# B&R Automation Studio project A2019059_Linka_Power_CP
Automation Studio 4.10.3.60 SP; technology packages: mapp 5.15.0, mappCockpit 5.15.0, mappMotion 5.15.1, mappView 5.15.1

## Configuration Config1

CPU 5PC900.TS17-00, AutomationRuntime B4.91, Build 6.3.0, Safety 1.10, Vc 

### Task classes (Cpu.sw)
```
Cyclic#1 (cycle 4000 us, tolerance 0 us):
  RiadenieSe <- RiadenieServ.RiadenieServ.prg
  P1_Skrutk1 <- Program.Pracovisko_1.P1_SkrutkovaciSet_M5.prg
  P1_Skrutk2 <- Program.Pracovisko_1.P1_SkrutkovaciSet_M4.prg
  P1_Skrutko <- Program.Pracovisko_1.P1_SkrutkovaciSet_K30.prg
  P2_Skrutko <- Program.Pracovisko_2.P2_SkrutkovaciSet_MaticaM4.prg
  P2_Skrutk2 <- Program.Pracovisko_2.P2_SkrutkovaciSet_M5.prg
  P2_Skrutk3 <- Program.Pracovisko_2.P2_SkrutkovaciSet_M6.prg
  P2_Skrutk1 <- Program.Pracovisko_2.P2_SkrutkovaciSet_M4.prg
  P3_Skrutk1 <- Program.Pracovisko_3.P3_SkrutkovaciSet_M5.prg
  P3_Skrutko <- Program.Pracovisko_3.P3_SkrutkovaciSet_K40.prg
  CAM_12 <- (binary)
  CAM_11 <- (binary)
  CAM_14 <- (binary)
  CAM_5 <- (binary)
  CAM_7 <- (binary)
  CAM_1 <- (binary)
  CAM_3 <- (binary)
  CAM_2 <- (binary)
  CAM_9 <- (binary)
  CAM_8 <- (binary)
  CAM_10 <- (binary)
  CAM_17 <- (binary)
  CAM_4 <- (binary)
  CAM_6 <- (binary)
  CAM_13 <- (binary)
  CAM_16 <- (binary)
  CAM_15 <- (binary)
  CAM1 <- (binary)
Cyclic#2 (cycle 8000 us, tolerance 0 us):
  TaktimePra <- MeranieTaktimePracovisk.TaktimeVytah_ST1.prg
  TaktimeSro <- MeranieTaktimePracovisk.TaktimeSrobovanie_ST2.prg
  TaktimeZak <- MeranieTaktimePracovisk.TaktimeZaklTesnenia_ST3.prg
  TaktimeMat <- MeranieTaktimePracovisk.TaktimeMaticovacka_ST4.prg
  TaktimeSr1 <- MeranieTaktimePracovisk.TaktimeSrobovanie_ST5.prg
  TaktimeZva <- MeranieTaktimePracovisk.TaktimeZvaranie_ST6.prg
  Taktime_Sr <- MeranieTaktimePracovisk.Taktime_Srobovanie_ST7.prg
  Taktime_Le <- MeranieTaktimePracovisk.Taktime_LeakageTestA_ST8A.prg
  Taktime_L1 <- MeranieTaktimePracovisk.Taktime_LeakageTestB_ST8B.prg
  Taktime_Fu <- MeranieTaktimePracovisk.Taktime_FunkcnyTestA_ST9A.prg
  Taktime_F1 <- MeranieTaktimePracovisk.Taktime_FunkcnyTestB_ST9B.prg
  Taktime_Et <- MeranieTaktimePracovisk.Taktime_Etiketovacka_ST9.prg
  Taktime_Vy <- MeranieTaktimePracovisk.Taktime_Vytah_ST10.prg
  FTP_CAM1 <- OdosielanieFotiek.FTP_CAM1.prg
  FTP_CAM2 <- OdosielanieFotiek.FTP_CAM2.prg
  FTP_CAM4 <- OdosielanieFotiek.FTP_CAM4.prg
  FTP_CAM6 <- OdosielanieFotiek.FTP_CAM6.prg
  FTP_CAM9 <- OdosielanieFotiek.FTP_CAM9.prg
  FTP_CAM10 <- OdosielanieFotiek.FTP_CAM10.prg
  FTP_CAM11 <- OdosielanieFotiek.FTP_CAM11.prg
  FTP_CAM12 <- OdosielanieFotiek.FTP_CAM12.prg
  FTP_CAM13 <- OdosielanieFotiek.FTP_CAM13.prg
  FTP_CAM15 <- OdosielanieFotiek.FTP_CAM15.prg
  FTP_CAM16 <- OdosielanieFotiek.FTP_CAM16.prg
  FTP_CAM17 <- OdosielanieFotiek.FTP_CAM17.prg
  FTP_DMP_CA <- OdosielanieFotiek.FTP_DMP_CAM1.prg
  FTP_DMP_C1 <- OdosielanieFotiek.FTP_DMP_CAM2.prg
  FTP_DMP_C2 <- OdosielanieFotiek.FTP_DMP_CAM3.prg
  FTP_DMP_C3 <- OdosielanieFotiek.FTP_DMP_CAM4.prg
  FTP_DMP_C4 <- OdosielanieFotiek.FTP_DMP_CAM5.prg
  FTP_DMP_C5 <- OdosielanieFotiek.FTP_DMP_CAM6.prg
  FTP_DMP_C6 <- OdosielanieFotiek.FTP_DMP_CAM7.prg
  FTP_DMP_C7 <- OdosielanieFotiek.FTP_DMP_CAM8.prg
  FTP_DMP_C8 <- OdosielanieFotiek.FTP_DMP_CAM9.prg
  FTP_DMP_C9 <- OdosielanieFotiek.FTP_DMP_CAM10.prg
  FTP_DMP_10 <- OdosielanieFotiek.FTP_DMP_CAM11.prg
  FTP_DMP_11 <- OdosielanieFotiek.FTP_DMP_CAM12.prg
  FTP_DMP_12 <- OdosielanieFotiek.FTP_DMP_CAM13.prg
  FTP_DMP_13 <- OdosielanieFotiek.FTP_DMP_CAM14.prg
  FTP_DMP_14 <- OdosielanieFotiek.FTP_DMP_CAM15.prg
  FTP_DMP_15 <- OdosielanieFotiek.FTP_DMP_CAM16.prg
  FTP_DMP_16 <- OdosielanieFotiek.FTP_DMP_CAM17.prg
  Users_Pane <- Uzivatelia.Users_Panel1.prg
  Users_Pan1 <- Uzivatelia.Users_Panel2.prg
  Program12 <- Uzivatelia.Users_Panel3.prg
  Users_Main <- Uzivatelia.Users_Main.prg
Cyclic#3 (cycle 48000 us, tolerance 48000 us):
  P1_Vytah_S <- TracebilitySystem.P1_Vytah_ST1.prg
  Program2 <- TracebilitySystem.P1_Srobovanie_ST2.prg
  Program3 <- TracebilitySystem.P2_ZakladacTesnenia_ST3.prg
  Program4 <- TracebilitySystem.P2_Maticovacka_ST4.prg
  Program5 <- TracebilitySystem.P2_Srobovanie_ST5.prg
  Program6 <- TracebilitySystem.P2_Zvaranie_ST6.prg
  Program7 <- TracebilitySystem.P3_Srobovanie_ST7.prg
  Program8 <- TracebilitySystem.P3_LeakageTestA_ST8A.prg
  Program9 <- TracebilitySystem.P3_LeakageTestB_ST8B.prg
  Program10 <- TracebilitySystem.P4_Etiketovacka_ST9.prg
  Program11 <- TracebilitySystem.P4_Vytah_ST10.prg
  LimitneSni <- RiadenieServ.LimitneSnimace.prg
  P4_StoperF <- Program.Pracovisko_4.P4_StoperFunkcnyTestA.prg
  P4_Stoper1 <- Program.Pracovisko_4.P4_StoperFunkcnyTestB.prg
  P3_Srobova <- Program.Pracovisko_3.P3_Srobovanie.prg
  Blikanie10 <- Blikace.Blikanie100ms.prg
Cyclic#4:
  Blikanie20 <- Blikace.Blikanie200ms.prg
  RFID_Prg <- Uzivatelia.RFID_Prg.prg
  P1_Main <- Program.Pracovisko_1.P1_Main.prg
  P1_Dopravn <- Program.Pracovisko_1.P1_Dopravniky.prg
  P1_SpodnyS <- Program.Pracovisko_1.P1_SpodnyStoper.prg
  P1_Akumula <- Program.Pracovisko_1.P1_AkumulacnyStoper.prg
  P1_Ovlada1 <- Program.Pracovisko_1.P1_OvladanieSafety.prg
  P2_Main <- Program.Pracovisko_2.P2_Main.prg
  P2_Dopravn <- Program.Pracovisko_2.P2_Dopravniky.prg
  P2_Akumula <- Program.Pracovisko_3.P3_VstupnyStoper.prg
  P2_Ovlada1 <- Program.Pracovisko_2.P2_OvladanieSafety.prg
  P3_Main <- Program.Pracovisko_3.P3_Main.prg
  P3_Dopravn <- Program.Pracovisko_3.P3_Dopravniky.prg
  P3_SpodnyS <- Program.Pracovisko_3.P3_SpodnyStoper.prg
  P3_Akumula <- Program.Pracovisko_3.P3_AkumulacnyStoper.prg
  P3_Ovlada1 <- Program.Pracovisko_3.P3_OvladanieSafety.prg
  P4_Main <- Program.Pracovisko_4.P4_Main.prg
  P4_Dopravn <- Program.Pracovisko_4.P4_Dopravniky.prg
  P4_Ovlada1 <- Program.Pracovisko_4.P4_OvladanieSafety.prg
  DatumCasPL <- DatumCasPLC.DatumCasPLC.prg
  Main <- Program.Linka.Main.prg
  OvladanieS <- Program.Linka.OvladanieSafety.prg
  UkladacieB <- UkladacieBuffery.UkladacieBuffery.prg
Cyclic#5 (cycle 248000 us, tolerance 248000 us):
  P1_Ovlada2 <- Program.Linka.OvladanieVizu.prg
  P1_Ovladan <- Program.Pracovisko_1.P1_OvladanieVizu.prg
  P2_Ovladan <- Program.Pracovisko_2.P2_OvladanieVizu.prg
  P3_Ovladan <- Program.Pracovisko_3.P34_OvladanieVizu.prg
  P1_Remanen <- RemanentnePremenne.P1_RemanentnePremenne.prg
  Remanentne <- RemanentnePremenne.P2_RemanentnePremenne.prg
  P34_Remane <- RemanentnePremenne.P34_RemanentnePremenne.prg
  Blikanie50 <- Blikace.Blikanie500ms.prg
Cyclic#6:
  Blikanie1s <- Blikace.Blikanie1s.prg
Cyclic#8 (cycle 8000 us, tolerance 8000 us):
  P1_Alarmy <- Alarmy.P1_Alarmy.prg
  P2_Alarmy <- Alarmy.P2_Alarmy.prg
  P34_Alarmy <- Alarmy.P34_Alarmy.prg
  P1_Vytah <- Program.Pracovisko_1.P1_Vytah.prg
  P1_Srobova <- Program.Pracovisko_1.P1_Srobovanie.prg
  P1_StoperS <- Program.Pracovisko_1.P1_StoperSrobovania.prg
  P1_Robot <- Program.Pracovisko_1.P1_Robot.prg
  P2_Zaklada <- Program.Pracovisko_2.P2_ZakladacTesnenia.prg
  P2_StoperZ <- Program.Pracovisko_2.P2_StoperZaklTesnenia.prg
  P2_StoperM <- Program.Pracovisko_2.P2_StoperMaticovacky.prg
  P2_Srobova <- Program.Pracovisko_2.P2_Srobovanie.prg
  P2_StoperS <- Program.Pracovisko_2.P2_StoperSrobovania.prg
  P2_Robot <- Program.Pracovisko_2.P2_Robot.prg
  P2_Zvarani <- Program.Pracovisko_2.P2_Zvaranie.prg
  P2_Cisteni <- Program.Pracovisko_2.P2_Cistenie.prg
  P2_Stoper1 <- Program.Pracovisko_2.P2_StoperZvarania.prg
  P3_StoperS <- Program.Pracovisko_3.P3_StoperSrobovania.prg
  P3_StoperL <- Program.Pracovisko_3.P3_StoperLeakageTestA.prg
  P3_Stoper1 <- Program.Pracovisko_3.P3_StoperLeakageTestB.prg
  P4_StoperE <- Program.Pracovisko_4.P4_StoperEtiketovacky.prg
  P4_Vytah <- Program.Pracovisko_4.P4_Vytah.prg
DataObjects: McAcpSys, assl1
Binaries: arsvcreg, udbdef, mvLoader, TCData, FWRules, mCoWebSc, mcacpdrv, McAcpSim, mcprofgen, TCLang, arflatprv, arcoal, ashwd, ashwac, Settings, User, sysconf, asfw, arconfig, asnxdb1, iomap, Role, Config_3, Config_1, Config, Config_2, Config_4, Config_5, Config_6, Config_7, Config_8, Config_9, Config_15, Config_14, TC, asiol4, asiol10, asiol3, asiol1, asiol2, Config_20, Config_19, Config_18, asiol5, Config_21, asiol6, asiol7, Config_23, Config_22, asiol9, asiol8, Config_10, asnxdb2, TraceConfi, Users, Config_13, Config_11, Config_12, Config_17, Config_16, asnxdb3
Libraries: CoTrace, AsZip, FileIO, runtime, AsBrStr, sys_lib, dvframe, AsUSB, standard, asstring, SC, AxisLib, MpBase, MpAlarmX, astime, MpRecipe, AsSafety, DataObj, AsXml, MpServer, AsBrWStr, AsIODiag, AsHttp, AsMem, AsMath, AsTCP, AsIecCon, IecCheck, MpAxis, McAxis, McBase, McAcpAx, McStpAx, McAcpPar, AtlasCopco, SKTcp, RFID, asio, asioacc, powerlnk, aruser, arssl, asepl, aseth, ashw, arcert
```

### Hardware
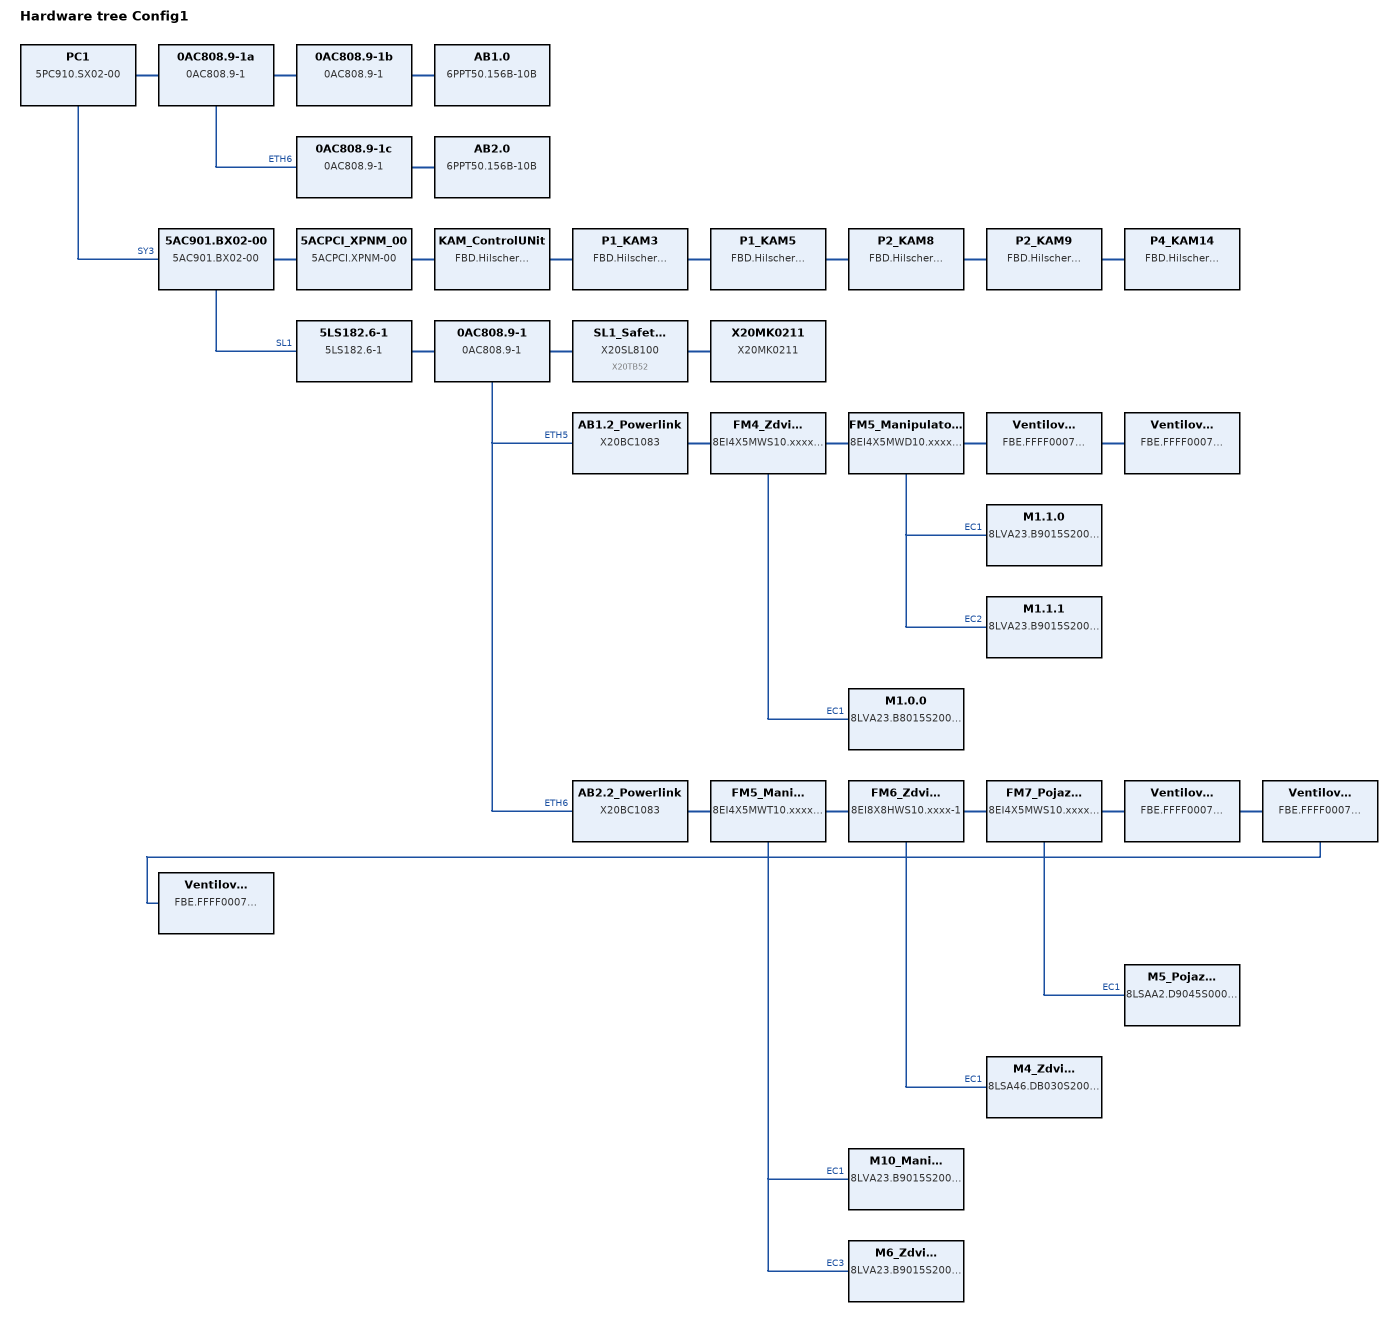
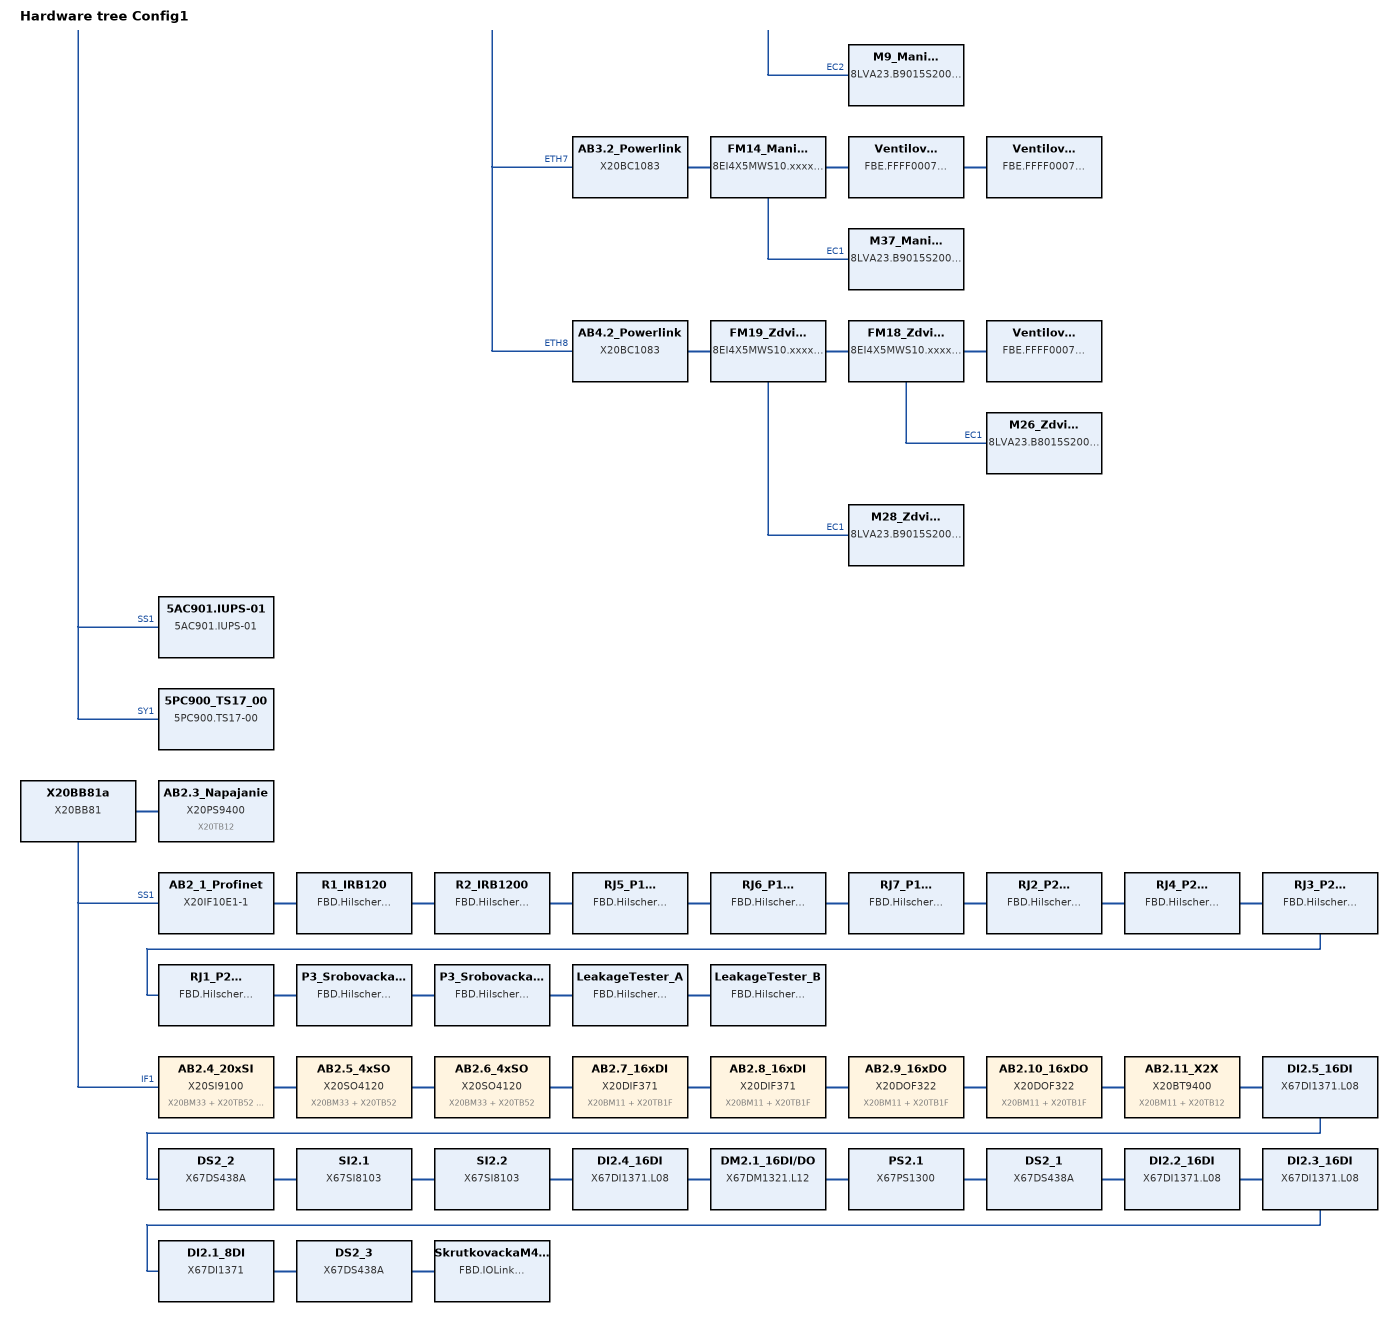
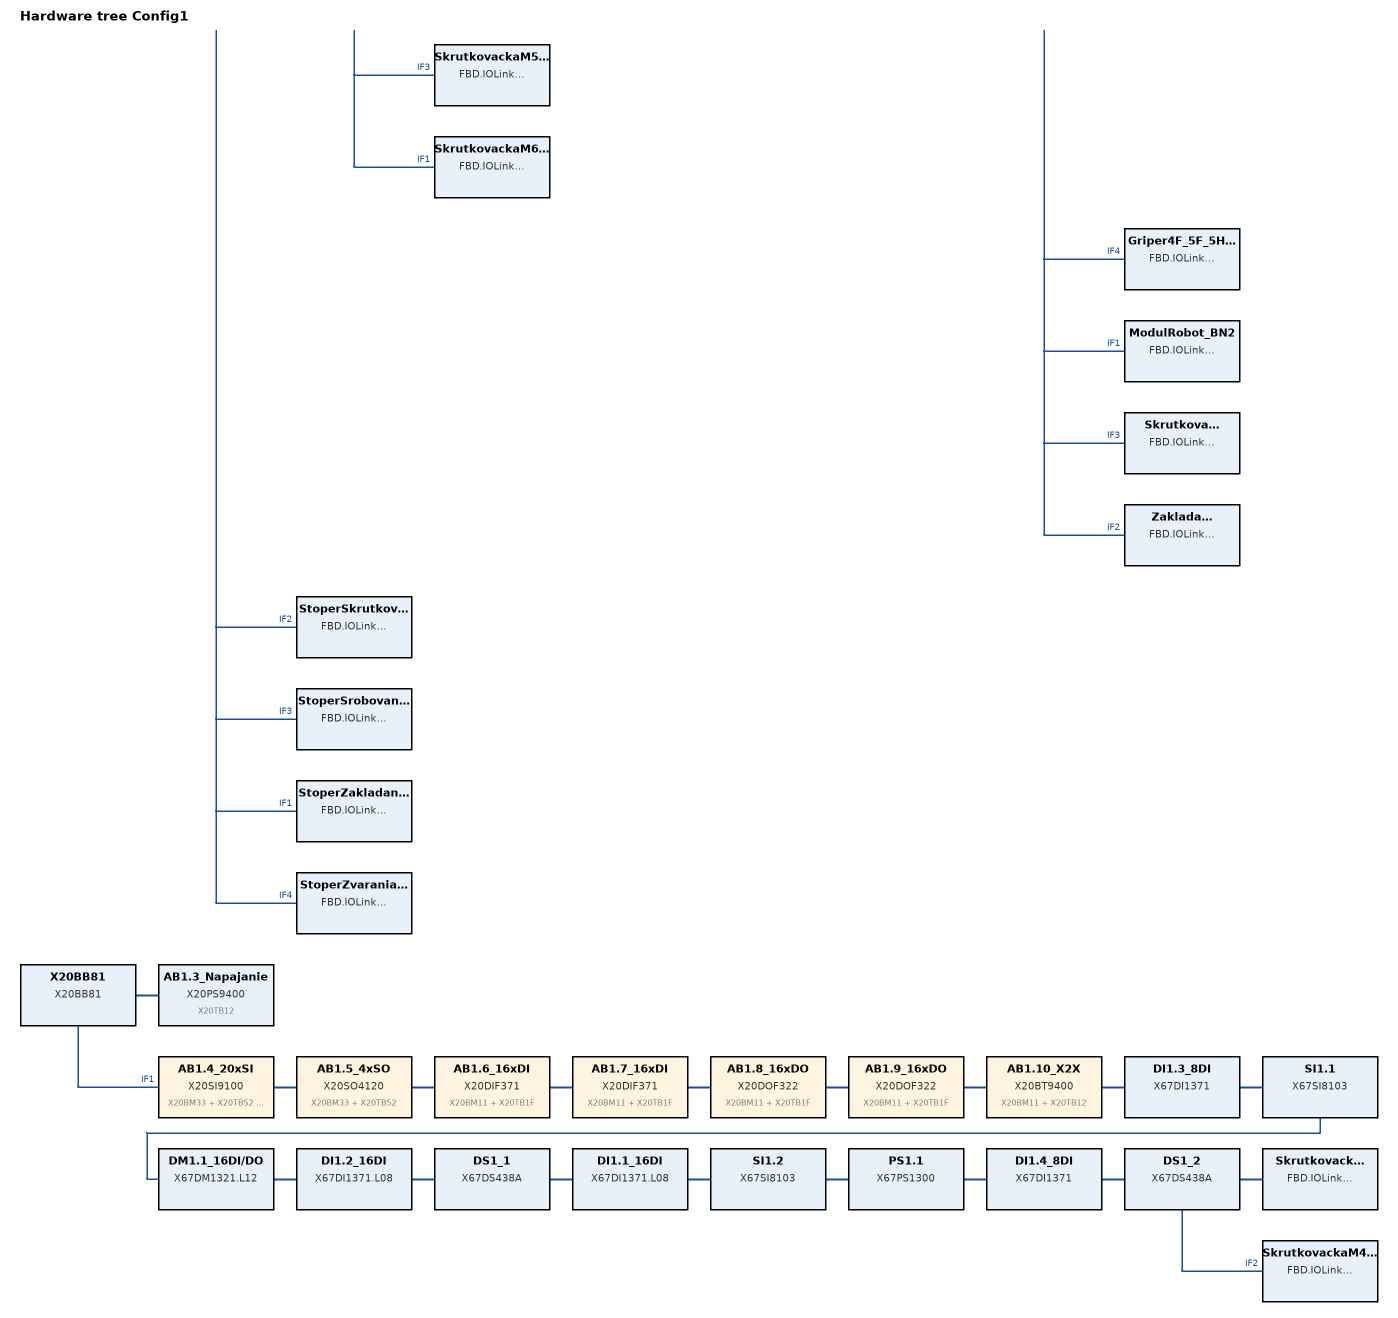
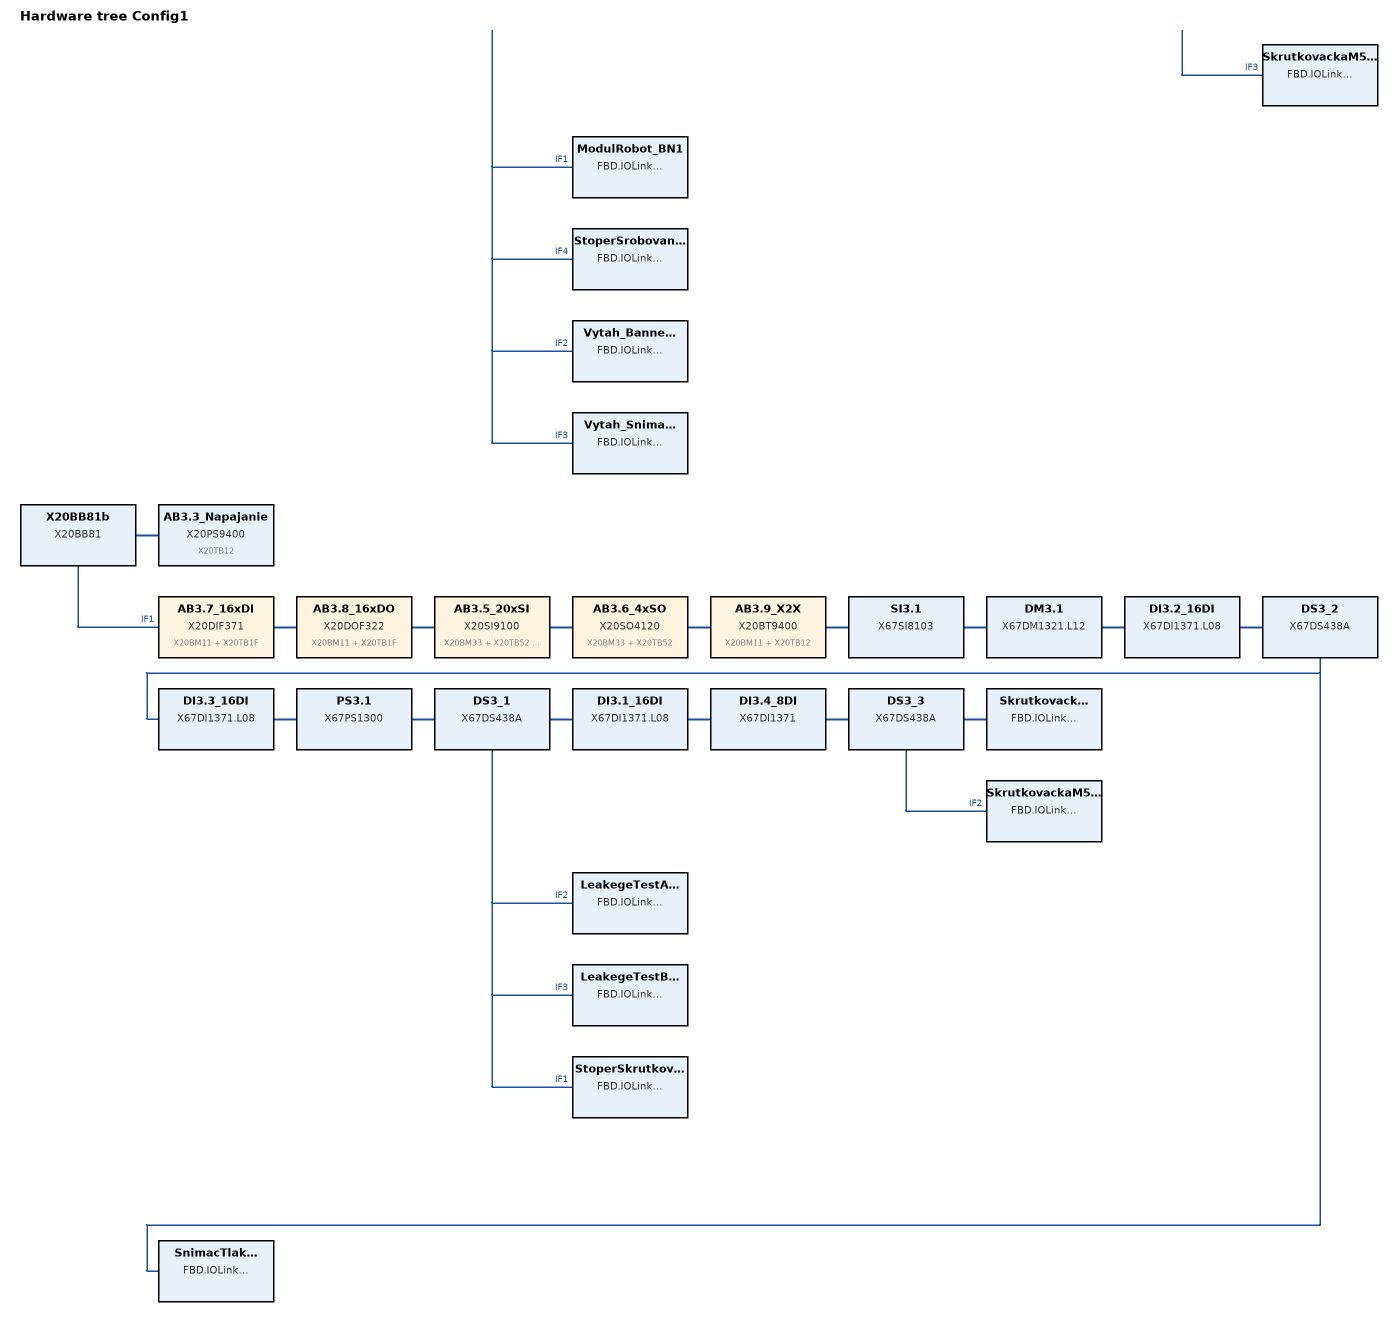
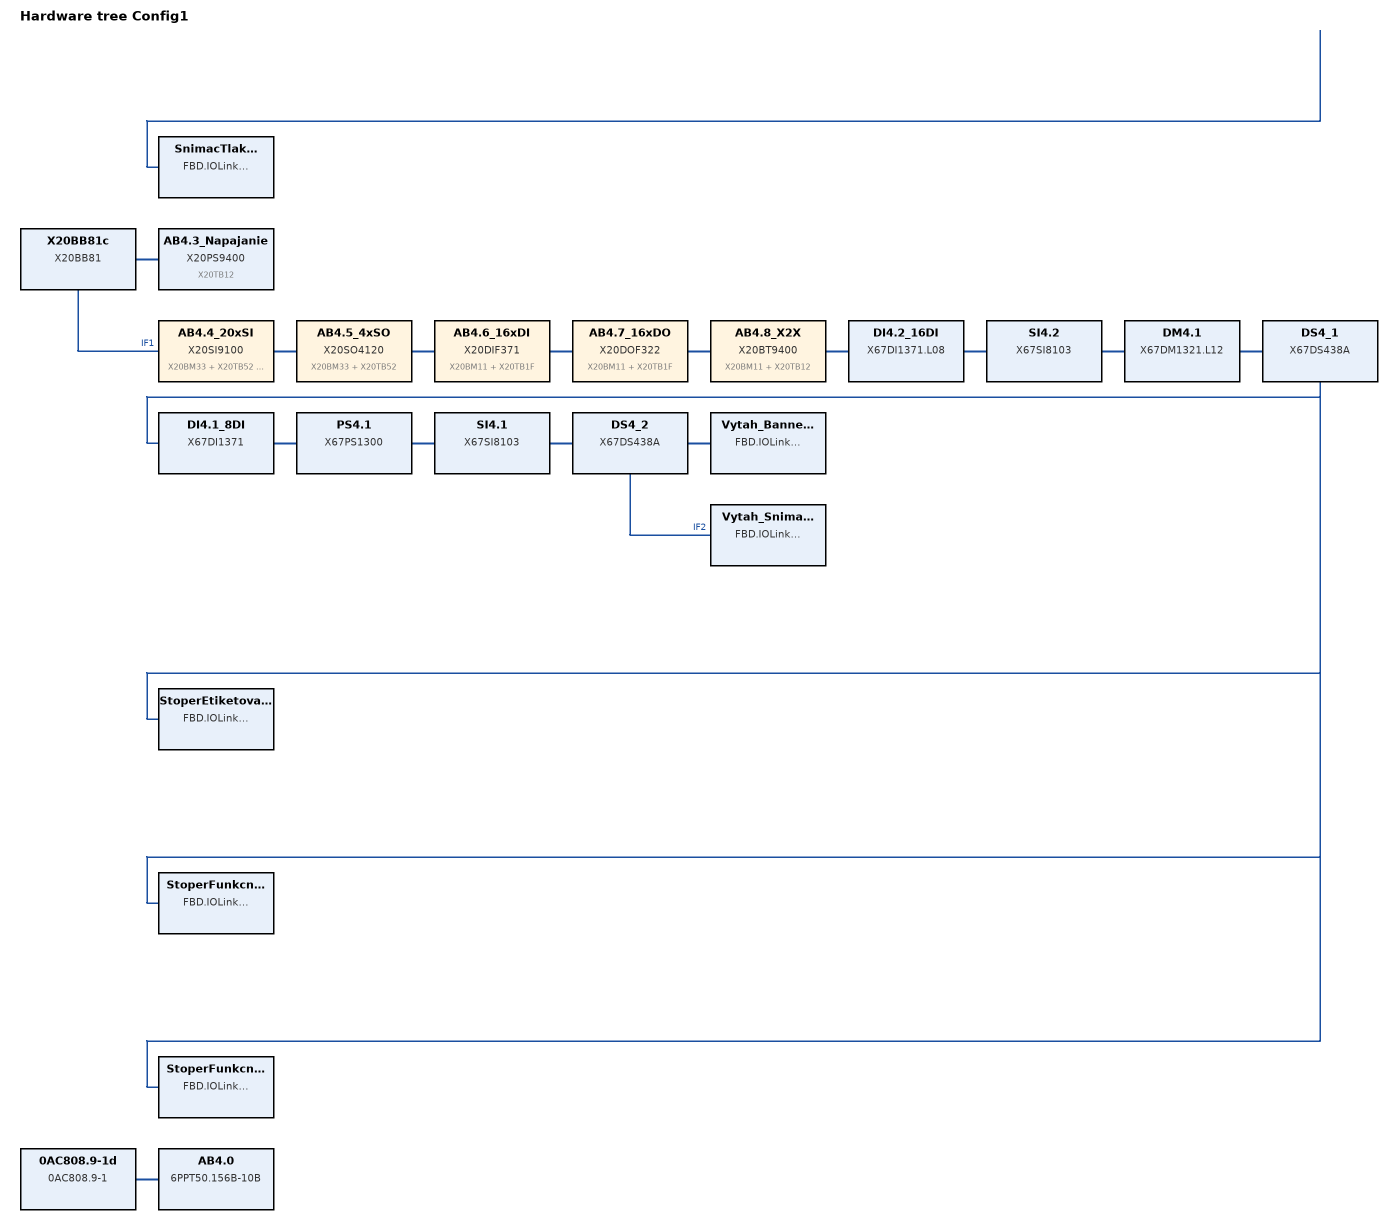
```
0AC808.9-1 : 0AC808.9-1 v1.0.0.0  [ETH1 -> 5LS182.6-1.IF1 [Cable Type=PowerlinkCable, Length=10, Version=1.0.0.3]; ETH2 -> SL1_SafetyMaster.PLK1 [Cable Type=PowerlinkCable, Length=10, Version=1.0.0.3]; ETH5 -> AB1.2_Powerlink.PLK1 [Cable Type=PowerlinkCable, Length=10, Version=1.0.0.3]; ETH6 -> AB2.2_Powerlink.PLK1 [Cable Type=PowerlinkCable, Length=10, Version=1.0.0.3]; ETH7 -> AB3.2_Powerlink.PLK1 [Cable Type=PowerlinkCable, Length=10, Version=1.0.0.3]; ETH8 -> AB4.2_Powerlink.PLK1 [Cable Type=PowerlinkCable, Length=10, Version=1.0.0.3]]
0AC808.9-1a : 0AC808.9-1 v1.0.0.0  [ETH1 -> PC1.IF3 [Cable Type=PowerlinkCable, Length=10, Version=1.0.0.3]; ETH5 -> 0AC808.9-1b.ETH1 [Cable Type=PowerlinkCable, Length=10, Version=1.0.0.3]; ETH6 -> 0AC808.9-1c.ETH1 [Cable Type=PowerlinkCable, Length=10, Version=1.0.0.3]; ETH8 -> 0AC808.9-1d.ETH8 [Cable Type=PowerlinkCable, Length=10, Version=1.0.0.3]]
0AC808.9-1b : 0AC808.9-1 v1.0.0.0  [ETH1 -> 0AC808.9-1a.ETH5 [Cable Type=PowerlinkCable, Length=10, Version=1.0.0.3]; ETH5 -> AB1.0.ETH1 [Cable Type=PowerlinkCable, Length=10, Version=1.0.0.3]]
0AC808.9-1c : 0AC808.9-1 v1.0.0.0  [ETH1 -> 0AC808.9-1a.ETH6 [Cable Type=PowerlinkCable, Length=10, Version=1.0.0.3]; ETH5 -> AB2.0.ETH1 [Cable Type=PowerlinkCable, Length=10, Version=1.0.0.3]]
0AC808.9-1d : 0AC808.9-1 v1.0.0.0  [ETH5 -> AB4.0.ETH1 [Cable Type=PowerlinkCable, Length=10, Version=1.0.0.3]; ETH8 -> 0AC808.9-1a.ETH8 [Cable Type=PowerlinkCable, Length=10, Version=1.0.0.3]]
5AC901.BX02-00 : 5AC901.BX02-00 v1.0.1.0  [SY -> PC1.SY3]
5AC901.IUPS-01 : 5AC901.IUPS-01 v1.3.1.0  [SS -> PC1.SS1]
  Supervision = off
5ACPCI_XPNM_00 : 5ACPCI.XPNM-00 v1.3.1.0  [SL -> 5AC901.BX02-00.SL2]
  Connector IF1:
    DtmId = 5eec11f9-fea1-40a1-ae00-7a0d8004f8c3
  ConfigFile = 5ACPCI_XPNM_00.dtm
  ConfigModule = asnxdb1
  CycleTime = 2000
5LS182.6-1 : 5LS182.6-1 v1.5.0.0  [SL -> 5AC901.BX02-00.SL1]
  Connector IF1:
    MtuSize = 800
    DNAConfiguration = manual
  Supervision = off
5PC900_TS17_00 : 5PC900.TS17-00 v2.1.0.0  [SY -> PC1.SY1]
  ConfigurationID = A2019059_Linka_Power_CP_Config1
  UserPartitionSize = 500
  UserRamDevice = PCI.1.LS182.SRAM
  UserRamSize = 10000
  RemMemDevice = PCI.1.LS182.SRAM
  RemMemSize = 54000
  PermanentPvSize = 20000
  RemanentGlobalPvSize = 4096
  VolatileGlobalPvSize = 300000
  EnableUsbRemoteInstall = 1
  RebootReset = 1
  TimerDeviceType = EPLX2X
  TimerDevice = 5LS182.6-1.IF1
  TaskClassIdleTime = 4000
  Cyclic1Duration = 4000
  Cyclic1Tolerance = 0
  Cyclic2Duration = 8000
  Cyclic2Tolerance = 0
  Cyclic3Duration = 48000
  Cyclic3Tolerance = 48000
  Cyclic5Duration = 248000
  Cyclic5Tolerance = 248000
  Cyclic8Duration = 8000
  Cyclic8Tolerance = 8000
  FileDevice1
  FileDeviceName1 = HDD_AlarmHistory
  FileDevicePath1 = F:\AlarmHistory
  FileDevice2
  FileDeviceName2 = HDD_RemPremenneP1
  FileDevicePath2 = F:\RemPremenneP1
  FileDevice3
  FileDeviceName3 = HDD_RemPremenneP2
  FileDevicePath3 = F:\RemPremenneP2
  FileDevice4
  FileDeviceName4 = HDD_RemPremenneP34
  FileDevicePath4 = F:\RemPremenneP34
  FileDevice5
  FileDeviceName5 = HDD_Users
  FileDevicePath5 = F:\Users
  FileDevice6
  FileDeviceName6 = HDD_Receptury
  FileDevicePath6 = F:\
  FileDevice7
  FileDeviceName7 = HDD_Audit
  FileDevicePath7 = F:\Audit
  FileDevice8
  FileDeviceName8 = HDD_Fotky
  FileDevicePath8 = F:\Kamery
  EthernetDefaultGateway = 192.168.122.1
  ActivateDns = 1
  DnsDefaultDomain = trst.prod
  DnsServer1 = 192.168.106.2
  FtpUser1
  FtpUsername1 = admin
  FtpUserPassword1 = txdC8JhjKtiQQqp7w9HbsY490GQe4kZyg7V65nMEvxA=
  FtpUserSalt1 = 0zleUdVK
  FTPAccessRight1 = 0
  ActivateDtmServer = 1
  ActivateOpcUa = 1
  OpcUa_Security_AdminRole = 
  OpcUaLimitsMaxSessions = 100
  OpcUaLimitsMaxPublish = 50
  OpcUaLimitsMaxBrowseContinuationPoints = 50
  OpcUa_Limits_MaxSubscriptionsPerSession = 30000
  OpcUa_Limits_MonitoredItemsPerSubscription = 5000
  OpcUaMaxSubsItemQueueSize = 5000
  OpcUaMaxSubsEventQueueSize = 5000
  OpcUaInformationModels_PV_Version = 1
  ActivateHypervisor = 1
  ARembDramSizeInMb = 2048
AB1.0 : 6PPT50.156B-10B v1.3.6.0  [ETH1 -> 0AC808.9-1b.ETH5 [Cable Type=PowerlinkCable, Length=10, Version=1.0.0.3]]
  Terminal = true
  Startmode = 2
  Mode = Manual
  InternetAddress = 192.168.122.11
  Subnetmask = 255.255.255.0
  DefaultGateway = 192.168.122.1
  ActivateNtpClient = 1
  NtpServer1 = 192.168.122.2
  TimeZone = 145
  PasswordVNC = 
  SelectedFavoriteWeb = 192.168.122.2:85/index.html?visuId=Vizu_P1
  BrowserVKeyboard = 0
  PasswordCIFS = 
  PasswordService = 
  VncRefreshRate = 100
AB1.10_X2X : X20BT9400 v1.3.0.0  [SS1 -> X20TB12d.SS; SL -> X20BM11h.SL1]
  Supervision = off
  PowerInfo = on
AB1.2_Powerlink : X20BC1083 v2.14.0.0  [PLK1 -> 0AC808.9-1.ETH5 (NodeNumber=11) [Cable Type=PowerlinkCable, Length=10, Version=1.0.0.3]; PLK2 -> FM4_ZdvihVytahu.PLK1 (NodeNumber=11) [Cable Type=PowerlinkCable, Length=10, Version=1.0.0.3]; SL -> X20BB81.SL1]
  Supervision = off
  ResponseTimeout = 50
AB1.3_Napajanie : X20PS9400 v1.7.0.0  [SS1 -> X20TB12.SS; PS -> X20BB81.PS1]
  Supervision = off
  PowerInfo = on
AB1.4_20xSI : X20SI9100 v1.10.12.0  [SS1 -> X20TB52a.SS; SS2 -> X20TB52b.SS; SL -> X20BM33.SL1]
  Supervision = off
  SafeModuleID = 10
AB1.5_4xSO : X20SO4120 v1.10.11.0  [SS1 -> X20TB52i.SS; SL -> X20BM33d.SL1]
  Supervision = off
  PLCopenInfo = on
  SafeModuleID = 11
  DigitalOutput01 = viaSafeLOGIC
  DigitalOutput02 = viaSafeLOGIC
  DigitalOutput03 = viaSafeLOGIC
  DigitalOutput04 = viaSafeLOGIC
AB1.6_16xDI : X20DIF371 v1.2.0.0  [SS1 -> X20TB1F.SS; SL -> X20BM11.SL1]
  Supervision = off
AB1.7_16xDI : X20DIF371 v1.2.0.0  [SS1 -> X20TB1F1.SS; SL -> X20BM11a.SL1]
  Supervision = off
AB1.8_16xDO : X20DOF322 v1.5.0.0  [SS1 -> X20TB1F2.SS; SL -> X20BM11b.SL1]
  Supervision = off
AB1.9_16xDO : X20DOF322 v1.5.0.0  [SS1 -> X20TB1F3.SS; SL -> X20BM11c.SL1]
  Supervision = off
AB2.0 : 6PPT50.156B-10B v1.3.6.0  [ETH1 -> 0AC808.9-1c.ETH5 [Cable Type=PowerlinkCable, Length=10, Version=1.0.0.3]]
  Terminal = true
  Startmode = 2
  Mode = Manual
  InternetAddress = 192.168.122.21
  Subnetmask = 255.255.255.0
  DefaultGateway = 192.168.122.1
  ActivateNtpClient = 1
  NtpServer1 = 192.168.122.2
  TimeZone = 145
  PasswordVNC = 
  SelectedFavoriteWeb = 192.168.122.2:85/index.html?visuId=Vizu_P2
  BrowserVKeyboard = 0
  PasswordCIFS = 
  PasswordService = 
  VncRefreshRate = 100
AB2.10_16xDO : X20DOF322 v1.5.0.0  [SS1 -> X20TB1F9.SS; SL -> X20BM11m.SL1]
  Supervision = off
AB2.11_X2X : X20BT9400 v1.3.0.0  [SS1 -> X20TB12e.SS; SL -> X20BM11i.SL1]
  Supervision = off
  PowerInfo = on
AB2.2_Powerlink : X20BC1083 v2.14.0.0  [PLK1 -> 0AC808.9-1.ETH6 (NodeNumber=21) [Cable Type=PowerlinkCable, Length=10, Version=1.0.0.3]; PLK2 -> FM5_ManipSrobovacky_ZdvihZvarania.PLK1 (NodeNumber=21) [Cable Type=PowerlinkCable, Length=10, Version=1.0.0.3]; SL -> X20BB81a.SL1]
  Supervision = off
  ResponseTimeout = 50
AB2.3_Napajanie : X20PS9400 v1.7.0.0  [SS1 -> X20TB12a.SS; PS -> X20BB81a.PS1]
  Supervision = off
  PowerInfo = on
AB2.4_20xSI : X20SI9100 v1.10.12.0  [SS1 -> X20TB52c.SS; SS2 -> X20TB52d.SS; SL -> X20BM33a.SL1]
  Supervision = off
  SafeModuleID = 20
AB2.5_4xSO : X20SO4120 v1.10.11.0  [SS1 -> X20TB52j.SS; SL -> X20BM33e.SL1]
  Supervision = off
  PLCopenInfo = on
  SafeModuleID = 21
  DigitalOutput01 = viaSafeLOGIC
  DigitalOutput02 = viaSafeLOGIC
  DigitalOutput03 = viaSafeLOGIC
  DigitalOutput04 = viaSafeLOGIC
AB2.6_4xSO : X20SO4120 v1.10.11.0  [SS1 -> X20TB52k.SS; SL -> X20BM33h.SL1]
  Supervision = off
  PLCopenInfo = on
  SafeModuleID = 22
  DigitalOutput01 = viaSafeLOGIC
  DigitalOutput02 = viaSafeLOGIC
  DigitalOutput03 = viaSafeLOGIC
  DigitalOutput04 = viaSafeLOGIC
AB2.7_16xDI : X20DIF371 v1.2.0.0  [SS1 -> X20TB1F4.SS; SL -> X20BM11d.SL1]
  Supervision = off
AB2.8_16xDI : X20DIF371 v1.2.0.0  [SS1 -> X20TB1F5.SS; SL -> X20BM11e.SL1]
  Supervision = off
AB2.9_16xDO : X20DOF322 v1.5.0.0  [SS1 -> X20TB1F8.SS; SL -> X20BM11l.SL1]
  Supervision = off
AB2_1_Profinet : X20IF10E1-1 v1.4.0.0  [SS -> X20BB81a.SS1]
  Connector IF1:
    DtmRef = FBDIF.Hilscher.PNIOControllerDTM2.NETX 100 RE/PNM
    DtmId = 08e46e45-e5af-4531-b20a-793914447b08
  ConfigFile = AB2_1_Profinet.dtm
  ConfigModule = asnxdb2
  CycleTime = 4000
AB3.2_Powerlink : X20BC1083 v2.14.0.0  [PLK1 -> 0AC808.9-1.ETH7 (NodeNumber=31) [Cable Type=PowerlinkCable, Length=10, Version=1.0.0.3]; PLK2 -> FM14_ManipSrobovacky.PLK1 (NodeNumber=31) [Cable Type=PowerlinkCable, Length=10, Version=1.0.0.3]; SL -> X20BB81b.SL1]
  Supervision = off
  ResponseTimeout = 50
AB3.3_Napajanie : X20PS9400 v1.7.0.0  [SS1 -> X20TB12b.SS; PS -> X20BB81b.PS1]
  Supervision = off
  PowerInfo = on
AB3.5_20xSI : X20SI9100 v1.10.12.0  [SS1 -> X20TB52e.SS; SS2 -> X20TB52f.SS; SL -> X20BM33b.SL1]
  Supervision = off
  SafeModuleID = 30
AB3.6_4xSO : X20SO4120 v1.10.11.0  [SS1 -> X20TB52l.SS; SL -> X20BM33f.SL1]
  Supervision = off
  PLCopenInfo = on
  SafeModuleID = 31
  DigitalOutput01 = viaSafeLOGIC
  DigitalOutput02 = viaSafeLOGIC
  DigitalOutput03 = viaSafeLOGIC
  DigitalOutput04 = viaSafeLOGIC
AB3.7_16xDI : X20DIF371 v1.2.0.0  [SS1 -> X20TB1F6.SS; SL -> X20BM11f.SL1]
  Supervision = off
AB3.8_16xDO : X20DOF322 v1.5.0.0  [SS1 -> X20TB1F7.SS; SL -> X20BM11g.SL1]
  Supervision = off
AB3.9_X2X : X20BT9400 v1.3.0.0  [SS1 -> X20TB12f.SS; SL -> X20BM11j.SL1]
  Supervision = off
AB4.0 : 6PPT50.156B-10B v1.3.6.0  [ETH1 -> 0AC808.9-1d.ETH5 [Cable Type=PowerlinkCable, Length=10, Version=1.0.0.3]]
  Terminal = true
  Startmode = 2
  Mode = Manual
  InternetAddress = 192.168.122.31
  Subnetmask = 255.255.255.0
  DefaultGateway = 192.168.122.1
  ActivateNtpClient = 1
  NtpServer1 = 192.168.122.2
  TimeZone = 145
  PasswordVNC = 
  SelectedFavoriteWeb = 192.168.122.2:85/index.html?visuId=Vizu_P34
  BrowserVKeyboard = 0
  PasswordCIFS = 
  PasswordService = 
  VncRefreshRate = 100
AB4.2_Powerlink : X20BC1083 v2.14.0.0  [PLK1 -> 0AC808.9-1.ETH8 (NodeNumber=41) [Cable Type=PowerlinkCable, Length=10, Version=1.0.0.3]; PLK2 -> FM19_ZdvihEtiketovacky.PLK1 (NodeNumber=41) [Cable Type=PowerlinkCable, Length=10, Version=1.0.0.3]; SL -> X20BB81c.SL1]
  Supervision = off
  ResponseTimeout = 50
AB4.3_Napajanie : X20PS9400 v1.7.0.0  [SS1 -> X20TB12c.SS; PS -> X20BB81c.PS1]
  Supervision = off
  PowerInfo = on
AB4.4_20xSI : X20SI9100 v1.10.12.0  [SS1 -> X20TB52g.SS; SS2 -> X20TB52h.SS; SL -> X20BM33c.SL1]
  Supervision = off
  SafeModuleID = 40
AB4.5_4xSO : X20SO4120 v1.10.11.0  [SS1 -> X20TB52m.SS; SL -> X20BM33g.SL1]
  Supervision = off
  PLCopenInfo = on
  SafeModuleID = 41
  DigitalOutput01 = viaSafeLOGIC
  DigitalOutput02 = viaSafeLOGIC
  DigitalOutput03 = viaSafeLOGIC
  DigitalOutput04 = viaSafeLOGIC
AB4.6_16xDI : X20DIF371 v1.2.0.0  [SS1 -> X20TB1F10.SS; SL -> X20BM11n.SL1]
  Supervision = off
AB4.7_16xDO : X20DOF322 v1.5.0.0  [SS1 -> X20TB1F11.SS; SL -> X20BM11o.SL1]
  Supervision = off
AB4.8_X2X : X20BT9400 v1.3.0.0  [SS1 -> X20TB12g.SS; SL -> X20BM11k.SL1]
  Supervision = off
  PowerInfo = on
DI1.1_16DI : X67DI1371.L08 v1.1.0.0  [X2X1 -> DS1_1.X2X2 [Cable Type=X2XCable, Length=10, Version=1.0.0.3]]
  Supervision = off
DI1.2_16DI : X67DI1371.L08 v1.1.0.0  [X2X1 -> DM1.1_16DI/DO.X2X2 [Cable Type=X2XCable, Length=10, Version=1.0.0.3]]
  Supervision = off
DI1.3_8DI : X67DI1371 v1.1.0.0  [X2X1 -> AB1.10_X2X.X2X1 [Cable Type=X2XCable, Length=10, Version=1.0.0.3]]
  Supervision = off
DI1.4_8DI : X67DI1371 v1.1.0.0  [X2X1 -> PS1.1.X2X2 [Cable Type=X2XCable, Length=10, Version=1.0.0.3]]
  Supervision = off
DI2.1_8DI : X67DI1371 v1.1.0.0  [X2X1 -> DI2.3_16DI.X2X2 [Cable Type=X2XCable, Length=10, Version=1.0.0.3]]
  Supervision = off
DI2.2_16DI : X67DI1371.L08 v1.1.0.0  [X2X1 -> DS2_1.X2X2 [Cable Type=X2XCable, Length=10, Version=1.0.0.3]]
  Supervision = off
DI2.3_16DI : X67DI1371.L08 v1.1.0.0  [X2X1 -> DI2.2_16DI.X2X2 [Cable Type=X2XCable, Length=10, Version=1.0.0.3]]
  Supervision = off
DI2.4_16DI : X67DI1371.L08 v1.1.0.0  [X2X1 -> SI2.2.X2X2 [Cable Type=X2XCable, Length=10, Version=1.0.0.3]]
  Supervision = off
DI2.5_16DI : X67DI1371.L08 v1.1.0.0  [X2X1 -> AB2.11_X2X.X2X1 [Cable Type=X2XCable, Length=10, Version=1.0.0.3]]
  Supervision = off
DI3.1_16DI : X67DI1371.L08 v1.1.0.0  [X2X1 -> DS3_1.X2X2 [Cable Type=X2XCable, Length=10, Version=1.0.0.3]]
  Supervision = off
DI3.2_16DI : X67DI1371.L08 v1.1.0.0  [X2X1 -> DM3.1.X2X2 [Cable Type=X2XCable, Length=10, Version=1.0.0.3]]
  Supervision = off
DI3.3_16DI : X67DI1371.L08 v1.1.0.0  [X2X1 -> DS3_2.X2X2 [Cable Type=X2XCable, Length=10, Version=1.0.0.3]]
  Supervision = off
DI3.4_8DI : X67DI1371 v1.1.0.0  [X2X1 -> DI3.1_16DI.X2X2 [Cable Type=X2XCable, Length=10, Version=1.0.0.3]]
  Supervision = off
DI4.1_8DI : X67DI1371 v1.1.0.0  [X2X1 -> DS4_1.X2X2 [Cable Type=X2XCable, Length=10, Version=1.0.0.3]]
  Supervision = off
DI4.2_16DI : X67DI1371.L08 v1.1.0.0  [X2X1 -> AB4.8_X2X.X2X1 [Cable Type=X2XCable, Length=10, Version=1.0.0.3]]
  Supervision = off
DM1.1_16DI/DO : X67DM1321.L12 v1.3.0.0  [X2X1 -> SI1.1.X2X2 [Cable Type=X2XCable, Length=10, Version=1.0.0.3]]
  Supervision = off
  Direction01 = output
  Direction03 = output
  Direction05 = output
  Direction07 = output
  Direction08 = output
  Direction09 = output
  Direction11 = output
  Direction13 = output
DM2.1_16DI/DO : X67DM1321.L12 v1.3.0.0  [X2X1 -> DI2.4_16DI.X2X2 [Cable Type=X2XCable, Length=10, Version=1.0.0.3]]
  Supervision = off
  Direction01 = output
  Direction03 = output
  Direction05 = output
  Direction07 = output
  Direction09 = output
  Direction11 = output
  Direction13 = output
  Direction15 = output
DM3.1 : X67DM1321.L12 v1.3.0.0  [X2X1 -> SI3.1.X2X2 [Cable Type=X2XCable, Length=10, Version=1.0.0.3]]
  Supervision = off
  Direction01 = output
  Direction03 = output
  Direction05 = output
  Direction07 = output
  Direction09 = output
DM4.1 : X67DM1321.L12 v1.3.0.0  [X2X1 -> SI4.2.X2X2 [Cable Type=X2XCable, Length=10, Version=1.0.0.3]]
  Supervision = off
  Direction01 = output
DS1_1 : X67DS438A v2.0.2.0  [X2X1 -> DI1.2_16DI.X2X2 [Cable Type=X2XCable, Length=10, Version=1.0.0.3]]
  DtmRef = FBD.BRIOLinkModuleDTM.DTMCore.X67DS438A
  DtmId = 5c77c125-df18-49d3-b5f3-4c14169cffef
  CommDtmId = 7d390211-d153-4b63-af3a-0fb4bd094c46
  RequiresDTMBuild = true
  ConfigFile = Communication.dtm
  ConfigModule = asiol2
  Supervision = off
  OperatingMode01 = Operate
  PDI_Enable01 = variousTypes
  PDI_DataType01_1 = USINT
  OperatingMode02 = Operate
  PDI_Enable02 = octetArray
  PDI_OctetSize02 = 2byte
  PDO_Enable02 = octetArray
  PDO_OctetSize02 = 10byte
  OperatingMode03 = Operate
  PDI_Enable03 = octetArray_DPS
  PDI_OctetSizeDPS03 = 10byte
  OperatingMode04 = Operate
  PDI_Enable04 = octetArray_DPS
  PDI_OctetSizeDPS04 = 10byte
DS1_2 : X67DS438A v2.0.2.0  [X2X1 -> DI1.4_8DI.X2X2 [Cable Type=X2XCable, Length=10, Version=1.0.0.3]]
  DtmRef = FBD.BRIOLinkModuleDTM.DTMCore.X67DS438A
  DtmId = e8efb28a-4369-4f6e-ba32-6070f12fc839
  CommDtmId = 7d390211-d153-4b63-af3a-0fb4bd094c46
  RequiresDTMBuild = true
  ConfigFile = Communication.dtm
  ConfigModule = asiol1
  Supervision = off
  OperatingMode01 = Operate
  PDI_Enable01 = variousTypes
  PDI_DataType01_1 = UINT
  OperatingMode02 = Operate
  PDI_Enable02 = variousTypes
  PDI_DataType02_1 = UINT
  OperatingMode03 = Operate
  PDI_Enable03 = variousTypes
  PDI_DataType03_1 = UINT
DS2_1 : X67DS438A v2.0.2.0  [X2X1 -> PS2.1.X2X2 [Cable Type=X2XCable, Length=10, Version=1.0.0.3]]
  DtmRef = FBD.BRIOLinkModuleDTM.DTMCore.X67DS438A
  DtmId = 6c6e43c7-21be-4bc5-b72d-9cc8aa168b62
  CommDtmId = 7d390211-d153-4b63-af3a-0fb4bd094c46
  RequiresDTMBuild = true
  ConfigFile = Communication.dtm
  ConfigModule = asiol3
  Supervision = off
  OperatingMode01 = Operate
  PDI_Enable01 = variousTypes
  PDI_DataType01_1 = USINT
  OperatingMode02 = Operate
  PDI_Enable02 = octetArray
  PDI_OctetSize02 = 2byte
  PDO_Enable02 = octetArray
  PDO_OctetSize02 = 10byte
  OperatingMode03 = Operate
  PDI_Enable03 = variousTypes
  PDI_DataType03_1 = UINT
  OperatingMode04 = Operate
  PDI_Enable04 = variousTypes
  PDI_DataType04_1 = UINT
DS2_2 : X67DS438A v2.0.2.0  [X2X1 -> DI2.5_16DI.X2X2 [Cable Type=X2XCable, Length=10, Version=1.0.0.3]]
  DtmRef = FBD.BRIOLinkModuleDTM.DTMCore.X67DS438A
  DtmId = 6dcf51c1-a267-435c-afe7-74a87a65980e
  CommDtmId = 7d390211-d153-4b63-af3a-0fb4bd094c46
  RequiresDTMBuild = true
  ConfigFile = Communication.dtm
  ConfigModule = asiol10
  Supervision = off
  OperatingMode01 = Operate
  PDI_Enable01 = octetArray_DPS
  PDI_OctetSizeDPS01 = 10byte
  OperatingMode02 = Operate
  PDI_Enable02 = octetArray_DPS
  PDI_OctetSizeDPS02 = 10byte
  OperatingMode03 = Operate
  PDI_Enable03 = octetArray_DPS
  PDI_OctetSizeDPS03 = 10byte
  OperatingMode04 = Operate
  PDI_Enable04 = octetArray_DPS
  PDI_OctetSizeDPS04 = 10byte
DS2_3 : X67DS438A v2.0.2.0  [X2X1 -> DI2.1_8DI.X2X2 [Cable Type=X2XCable, Length=10, Version=1.0.0.3]]
  DtmRef = FBD.BRIOLinkModuleDTM.DTMCore.X67DS438A
  DtmId = 340b556e-295f-4e6a-bd8b-75a070d42850
  CommDtmId = 7d390211-d153-4b63-af3a-0fb4bd094c46
  RequiresDTMBuild = true
  ConfigFile = Communication.dtm
  ConfigModule = asiol4
  Supervision = off
  OperatingMode01 = Operate
  PDI_Enable01 = variousTypes
  PDI_DataType01_1 = UINT
  OperatingMode02 = Operate
  PDI_Enable02 = variousTypes
  PDI_DataType02_1 = UINT
  OperatingMode03 = Operate
  PDI_Enable03 = variousTypes
  PDI_DataType03_1 = UINT
DS3_1 : X67DS438A v2.0.2.0  [X2X1 -> PS3.1.X2X2 [Cable Type=X2XCable, Length=10, Version=1.0.0.3]]
  DtmRef = FBD.BRIOLinkModuleDTM.DTMCore.X67DS438A
  DtmId = 9d23c650-c770-4c6e-b46f-8263eb440c8e
  CommDtmId = 7d390211-d153-4b63-af3a-0fb4bd094c46
  RequiresDTMBuild = true
  ConfigFile = Communication.dtm
  ConfigModule = asiol6
  Supervision = off
  OperatingMode01 = Operate
  PDI_Enable01 = octetArray_DPS
  PDI_OctetSizeDPS01 = 10byte
  OperatingMode02 = Operate
  PDI_Enable02 = octetArray_DPS
  PDI_OctetSizeDPS02 = 10byte
  OperatingMode03 = Operate
  PDI_Enable03 = octetArray_DPS
  PDI_OctetSizeDPS03 = 10byte
DS3_2 : X67DS438A v2.0.2.0  [X2X1 -> DI3.2_16DI.X2X2 [Cable Type=X2XCable, Length=10, Version=1.0.0.3]]
  DtmRef = FBD.BRIOLinkModuleDTM.DTMCore.X67DS438A
  DtmId = a7eb8fb6-db97-4afc-b9d3-8750693ebcbe
  CommDtmId = 7d390211-d153-4b63-af3a-0fb4bd094c46
  RequiresDTMBuild = true
  ConfigFile = Communication.dtm
  ConfigModule = asiol5
  Supervision = off
  OperatingMode01 = Operate
  PDI_Enable01 = variousTypes
  PDI_DataType01_1 = UINT
  OperatingMode02 = Operate
  PDI_Enable02 = variousTypes
  PDI_DataType02_1 = UINT
DS3_3 : X67DS438A v2.0.2.0  [X2X1 -> DI3.4_8DI.X2X2 [Cable Type=X2XCable, Length=10, Version=1.0.0.3]]
  DtmRef = FBD.BRIOLinkModuleDTM.DTMCore.X67DS438A
  DtmId = 368358d0-453a-4650-9d77-1e5a5bfd0086
  CommDtmId = 7d390211-d153-4b63-af3a-0fb4bd094c46
  RequiresDTMBuild = true
  ConfigFile = Communication.dtm
  ConfigModule = asiol7
  Supervision = off
  CycleEndEnable = on
  SyncInformationEnable = on
  OperatingMode01 = Operate
  PDI_Enable01 = variousTypes
  PDI_DataType01_1 = UINT
  OperatingMode02 = Operate
  PDI_Enable02 = variousTypes
  PDI_DataType02_1 = UINT
DS4_1 : X67DS438A v2.0.2.0  [X2X1 -> DM4.1.X2X2 [Cable Type=X2XCable, Length=10, Version=1.0.0.3]]
  DtmRef = FBD.BRIOLinkModuleDTM.DTMCore.X67DS438A
  DtmId = 812b7be7-ea90-49cd-bd0f-6922f0b365ce
  CommDtmId = 7d390211-d153-4b63-af3a-0fb4bd094c46
  RequiresDTMBuild = true
  ConfigFile = Communication.dtm
  ConfigModule = asiol8
  Supervision = off
  OperatingMode01 = Operate
  PDI_Enable01 = octetArray_DPS
  PDI_OctetSizeDPS01 = 10byte
  OperatingMode02 = Operate
  PDI_Enable02 = octetArray_DPS
  PDI_OctetSizeDPS02 = 10byte
  OperatingMode03 = Operate
  PDI_Enable03 = octetArray_DPS
  PDI_OctetSizeDPS03 = 10byte
DS4_2 : X67DS438A v2.0.2.0  [X2X1 -> SI4.1.X2X2 [Cable Type=X2XCable, Length=10, Version=1.0.0.3]]
  DtmRef = FBD.BRIOLinkModuleDTM.DTMCore.X67DS438A
  DtmId = 630fd496-1eda-4307-8763-f03027e0c3fb
  CommDtmId = 7d390211-d153-4b63-af3a-0fb4bd094c46
  RequiresDTMBuild = true
  ConfigFile = Communication.dtm
  ConfigModule = asiol9
  Supervision = off
  OperatingMode01 = Operate
  PDI_Enable01 = octetArray
  PDI_OctetSize01 = 2byte
  PDO_Enable01 = octetArray
  PDO_OctetSize01 = 10byte
  OperatingMode02 = Operate
  PDI_Enable02 = octetArray_DPS
  PDI_OctetSizeDPS02 = 10byte
FM14_ManipSrobovacky : 8EI4X5MWS10.xxxx-1 v2.3.1.1  [PLK1 -> AB3.2_Powerlink.PLK2 [Cable Type=PowerlinkCable, Length=10, Version=1.0.0.3]; PLK2 -> VentilovyTerminal_VT6.PLK1 [Cable Type=PowerlinkCable, Length=10, Version=1.0.0.3]; EC1 -> M37_ManipSrobovackyOsY.EC]
  ResponseTimeout = 50
  DriveConfiguration/Module:
    McAcoposTypeID = AcoposP3DConfig
    ActivateACOPOSSimulationOnPLC = 0
  DriveConfiguration/Encoder/EncoderX41:
    InterfaceType = EnDat
  DriveConfiguration/Channel[1]:
    License = 1
  DriveConfiguration/Channel[1]/RealAxis:
    AxisReference = gAxis_9
  DriveConfiguration/Channel[1]/RealAxis/MechanicalElements/Gearbox:
    InputIsReadOnly = 0
    Input = 1
    OutputIsReadOnly = 0
    Output = 1
  DriveConfiguration/Channel[1]/RealAxis/MechanicalElements/RotaryToLinearTransformation:
    ReferenceDistanceIsReadOnly = 0
    ReferenceDistance = 10  // Rozlíšenie - 10mm/otačku
  DriveConfiguration/Channel[1]/RealAxis/Controller:
    ModeIsReadOnly = 0
    Mode = PositionController
  DriveConfiguration/Channel[1]/RealAxis/Controller/Mode/Position:
    ProportionalGain = 535
    IntegrationTime = 0.0
    PredictionTime = 0.0004
    TotalDelayTime = 0.0004
  DriveConfiguration/Channel[1]/RealAxis/Controller/Mode/Speed:
    ProportionalGainIsReadOnly = 0
    ProportionalGain = 1.5
    IntegrationTimeIsReadOnly = 0
    IntegrationTime = 0.0
    FilterTimeIsReadOnly = 0
    FilterTime = 0.0
  DriveConfiguration/Channel[1]/RealAxis/Controller/Mode/LoopFilters:
    LoopFilter1 = NotUsed
    LoopFilter2 = NotUsed
    LoopFilter3 = NotUsed
  DriveConfiguration/Channel[1]/RealAxis/Homing:
    Mode = Direct
  DriveConfiguration/Channel[1]/RealAxis/Homing/Mode:
    Position = 0.0
    ReferencePulse = NotUsed
  DriveConfiguration/Channel[1]/RealAxis/Homing:
    RestorePositionVariable = 
  DriveConfiguration/Channel[1]/RealAxis/StopReaction:
    Quickstop = DecelerationLimit
    DriveError = DecelerationLimit
  DriveConfiguration/Channel[1]/RealAxis/MovementErrorLimits:
    PositionError = 1.0
    VelocityErrorMonitoring = Automatic1
  DriveConfiguration/Channel[1]/RealAxis:
    JerkFilter = NotUsed
  DriveConfiguration/Channel[1]/RealAxis/DigitalInputs/HomingSwitch:
    Source = NotUsed
    Level = High
  DriveConfiguration/Channel[1]/RealAxis/DigitalInputs/PositiveLimitSwitch:
    Source = NotUsed
    Level = High
  DriveConfiguration/Channel[1]/RealAxis/DigitalInputs/NegativeLimitSwitch:
    Source = NotUsed
    Level = High
  DriveConfiguration/Channel[1]/RealAxis/DigitalInputs/Trigger1:
    Source = X8Trigger1
    Level = High
  DriveConfiguration/Channel[1]/RealAxis/DigitalInputs/Trigger2:
    Source = X8Trigger2
    Level = High
  DriveConfiguration/Channel[1]/RealAxis/DigitalInputs/Quickstop:
    Input = Trigger2
  DriveConfiguration/Channel[1]/RealAxis/Simulation:
    SimulationModeOnPLC = SetValueGeneration
    SimulationModeOnACOPOS = NotUsed
FM18_ZdvihVytahu : 8EI4X5MWS10.xxxx-1 v2.3.1.1  [PLK1 -> FM19_ZdvihEtiketovacky.PLK2 [Cable Type=PowerlinkCable, Length=10, Version=1.0.0.3]; PLK2 -> VentilovyTerminal_VT8.PLK1 [Cable Type=PowerlinkCable, Length=10, Version=1.0.0.3]; EC1 -> M26_ZdvihVytahu.EC]
  ResponseTimeout = 50
  DriveConfiguration/Module:
    McAcoposTypeID = AcoposP3DConfig
    ActivateACOPOSSimulationOnPLC = 0
  DriveConfiguration/Encoder/EncoderX41:
    InterfaceType = EnDat
  DriveConfiguration/Channel[1]:
    License = 1
  DriveConfiguration/Channel[1]/RealAxis:
    AxisReference = gAxis_10
  DriveConfiguration/Channel[1]/RealAxis/MechanicalElements/Gearbox:
    InputIsReadOnly = 0
    Input = 1
    OutputIsReadOnly = 0
    Output = 1
  DriveConfiguration/Channel[1]/RealAxis/MechanicalElements/RotaryToLinearTransformation:
    ReferenceDistanceIsReadOnly = 0
    ReferenceDistance = 5  // Rozlíšenie - 5mm/otačku
  DriveConfiguration/Channel[1]/RealAxis/Controller:
    ModeIsReadOnly = 0
    Mode = PositionController
  DriveConfiguration/Channel[1]/RealAxis/Controller/Mode/Position:
    ProportionalGain = 420
    IntegrationTime = 0.0
    PredictionTime = 0.0004
    TotalDelayTime = 0.0004
  DriveConfiguration/Channel[1]/RealAxis/Controller/Mode/Speed:
    ProportionalGainIsReadOnly = 0
    ProportionalGain = 6.5
    IntegrationTimeIsReadOnly = 0
    IntegrationTime = 0.0
    FilterTimeIsReadOnly = 0
    FilterTime = 0.0
  DriveConfiguration/Channel[1]/RealAxis/Controller/Mode/LoopFilters:
    LoopFilter1 = NotUsed
    LoopFilter2 = NotUsed
    LoopFilter3 = NotUsed
  DriveConfiguration/Channel[1]/RealAxis/Homing:
    Mode = Direct
  DriveConfiguration/Channel[1]/RealAxis/Homing/Mode:
    Position = 0.0
    ReferencePulse = NotUsed
  DriveConfiguration/Channel[1]/RealAxis/Homing:
    RestorePositionVariable = 
  DriveConfiguration/Channel[1]/RealAxis/StopReaction:
    Quickstop = DecelerationLimit
    DriveError = DecelerationLimit
  DriveConfiguration/Channel[1]/RealAxis/MovementErrorLimits:
    PositionError = 1.0
    VelocityErrorMonitoring = Automatic1
  DriveConfiguration/Channel[1]/RealAxis:
    JerkFilter = NotUsed
  DriveConfiguration/Channel[1]/RealAxis/DigitalInputs/HomingSwitch:
    Source = NotUsed
    Level = High
  DriveConfiguration/Channel[1]/RealAxis/DigitalInputs/PositiveLimitSwitch:
    Source = NotUsed
    Level = High
  DriveConfiguration/Channel[1]/RealAxis/DigitalInputs/NegativeLimitSwitch:
    Source = NotUsed
    Level = High
  DriveConfiguration/Channel[1]/RealAxis/DigitalInputs/Trigger1:
    Source = X8Trigger1
    Level = High
  DriveConfiguration/Channel[1]/RealAxis/DigitalInputs/Trigger2:
    Source = X8Trigger2
    Level = High
  DriveConfiguration/Channel[1]/RealAxis/DigitalInputs/Quickstop:
    Input = Trigger2
  DriveConfiguration/Channel[1]/RealAxis/Simulation:
    SimulationModeOnPLC = SetValueGeneration
    SimulationModeOnACOPOS = NotUsed
FM19_ZdvihEtiketovacky : 8EI4X5MWS10.xxxx-1 v2.3.1.1  [PLK1 -> AB4.2_Powerlink.PLK2 [Cable Type=PowerlinkCable, Length=10, Version=1.0.0.3]; PLK2 -> FM18_ZdvihVytahu.PLK1 [Cable Type=PowerlinkCable, Length=10, Version=1.0.0.3]; EC1 -> M28_ZdvihEtiketovacky.EC]
  ResponseTimeout = 50
  DriveConfiguration/Module:
    McAcoposTypeID = AcoposP3DConfig
    ActivateACOPOSSimulationOnPLC = 0
  DriveConfiguration/Encoder/EncoderX41:
    InterfaceType = EnDat
  DriveConfiguration/Channel[1]:
    License = 1
  DriveConfiguration/Channel[1]/RealAxis:
    AxisReference = gAxis_11
  DriveConfiguration/Channel[1]/RealAxis/MechanicalElements/Gearbox:
    InputIsReadOnly = 0
    Input = 1
    OutputIsReadOnly = 0
    Output = 1
  DriveConfiguration/Channel[1]/RealAxis/MechanicalElements/RotaryToLinearTransformation:
    ReferenceDistanceIsReadOnly = 0
    ReferenceDistance = 10  // Rozlíšenie - 10mm/otačku
  DriveConfiguration/Channel[1]/RealAxis/Controller:
    ModeIsReadOnly = 0
    Mode = PositionController
  DriveConfiguration/Channel[1]/RealAxis/Controller/Mode/Position:
    ProportionalGain = 478
    IntegrationTime = 0.0
    PredictionTime = 0.0004
    TotalDelayTime = 0.0004
  DriveConfiguration/Channel[1]/RealAxis/Controller/Mode/Speed:
    ProportionalGainIsReadOnly = 0
    ProportionalGain = 3
    IntegrationTimeIsReadOnly = 0
    IntegrationTime = 0.0
    FilterTimeIsReadOnly = 0
    FilterTime = 0.0
  DriveConfiguration/Channel[1]/RealAxis/Controller/Mode/LoopFilters:
    LoopFilter1 = NotUsed
    LoopFilter2 = NotUsed
    LoopFilter3 = NotUsed
  DriveConfiguration/Channel[1]/RealAxis/Homing:
    Mode = Direct
  DriveConfiguration/Channel[1]/RealAxis/Homing/Mode:
    Position = 0.0
    ReferencePulse = NotUsed
  DriveConfiguration/Channel[1]/RealAxis/Homing:
    RestorePositionVariable = 
  DriveConfiguration/Channel[1]/RealAxis/StopReaction:
    Quickstop = DecelerationLimit
    DriveError = DecelerationLimit
  DriveConfiguration/Channel[1]/RealAxis/MovementErrorLimits:
    PositionError = 1.0
    VelocityErrorMonitoring = Automatic1
  DriveConfiguration/Channel[1]/RealAxis:
    JerkFilter = NotUsed
  DriveConfiguration/Channel[1]/RealAxis/DigitalInputs/HomingSwitch:
    Source = NotUsed
    Level = High
  DriveConfiguration/Channel[1]/RealAxis/DigitalInputs/PositiveLimitSwitch:
    Source = NotUsed
    Level = High
  DriveConfiguration/Channel[1]/RealAxis/DigitalInputs/NegativeLimitSwitch:
    Source = NotUsed
    Level = High
  DriveConfiguration/Channel[1]/RealAxis/DigitalInputs/Trigger1:
    Source = X8Trigger1
    Level = High
  DriveConfiguration/Channel[1]/RealAxis/DigitalInputs/Trigger2:
    Source = X8Trigger2
    Level = High
  DriveConfiguration/Channel[1]/RealAxis/DigitalInputs/Quickstop:
    Input = Trigger2
  DriveConfiguration/Channel[1]/RealAxis/Simulation:
    SimulationModeOnPLC = SetValueGeneration
    SimulationModeOnACOPOS = NotUsed
FM4_ZdvihVytahu : 8EI4X5MWS10.xxxx-1 v2.3.1.1  [PLK1 -> AB1.2_Powerlink.PLK2 [Cable Type=PowerlinkCable, Length=10, Version=1.0.0.3]; PLK2 -> FM5_ManipulatorSrobovacky.PLK1 [Cable Type=PowerlinkCable, Length=10, Version=1.0.0.3]; EC1 -> M1.0.0.EC]
  ResponseTimeout = 50
  DriveConfiguration/Module:
    McAcoposTypeID = AcoposP3DConfig
    ActivateACOPOSSimulationOnPLC = 0
  DriveConfiguration/Encoder/EncoderX41:
    InterfaceType = EnDat
  DriveConfiguration/Channel[1]:
    License = 1
  DriveConfiguration/Channel[1]/RealAxis:
    AxisReference = gAxis_6
  DriveConfiguration/Channel[1]/RealAxis/MechanicalElements/Gearbox:
    InputIsReadOnly = 0
    Input = 1
    OutputIsReadOnly = 0
    Output = 1
  DriveConfiguration/Channel[1]/RealAxis/MechanicalElements/RotaryToLinearTransformation:
    ReferenceDistanceIsReadOnly = 0
    ReferenceDistance = 5  // Rozlíšenie - 5mm/otačku
  DriveConfiguration/Channel[1]/RealAxis/Controller:
    ModeIsReadOnly = 0
    Mode = PositionController
  DriveConfiguration/Channel[1]/RealAxis/Controller/Mode/Position:
    ProportionalGain = 425
    IntegrationTime = 0.0
    PredictionTime = 0.0004
    TotalDelayTime = 0.0004
  DriveConfiguration/Channel[1]/RealAxis/Controller/Mode/Speed:
    ProportionalGainIsReadOnly = 0
    ProportionalGain = 4.6
    IntegrationTimeIsReadOnly = 0
    IntegrationTime = 0.0
    FilterTimeIsReadOnly = 0
    FilterTime = 0.0
  DriveConfiguration/Channel[1]/RealAxis/Controller/Mode/LoopFilters:
    LoopFilter1 = NotUsed
    LoopFilter2 = NotUsed
    LoopFilter3 = NotUsed
  DriveConfiguration/Channel[1]/RealAxis/Homing:
    Mode = Direct
  DriveConfiguration/Channel[1]/RealAxis/Homing/Mode:
    Position = 0.0
    ReferencePulse = NotUsed
  DriveConfiguration/Channel[1]/RealAxis/Homing:
    RestorePositionVariable = 
  DriveConfiguration/Channel[1]/RealAxis/StopReaction:
    Quickstop = DecelerationLimit
    DriveError = DecelerationLimit
  DriveConfiguration/Channel[1]/RealAxis/MovementErrorLimits:
    PositionError = 1.0
    VelocityErrorMonitoring = Automatic1
  DriveConfiguration/Channel[1]/RealAxis:
    JerkFilter = NotUsed
  DriveConfiguration/Channel[1]/RealAxis/DigitalInputs/HomingSwitch:
    Source = NotUsed
    Level = High
  DriveConfiguration/Channel[1]/RealAxis/DigitalInputs/PositiveLimitSwitch:
    Source = NotUsed
    Level = High
  DriveConfiguration/Channel[1]/RealAxis/DigitalInputs/NegativeLimitSwitch:
    Source = NotUsed
    Level = High
  DriveConfiguration/Channel[1]/RealAxis/DigitalInputs/Trigger1:
    Source = X8Trigger1
    Level = High
  DriveConfiguration/Channel[1]/RealAxis/DigitalInputs/Trigger2:
    Source = X8Trigger2
    Level = High
  DriveConfiguration/Channel[1]/RealAxis/DigitalInputs/Quickstop:
    Input = Trigger2
  DriveConfiguration/Channel[1]/RealAxis/Simulation:
    SimulationModeOnPLC = SetValueGeneration
    SimulationModeOnACOPOS = NotUsed
FM5_ManipSrobovacky_ZdvihZvarania : 8EI4X5MWT10.xxxx-1 v2.3.1.1  [PLK1 -> AB2.2_Powerlink.PLK2 [Cable Type=PowerlinkCable, Length=10, Version=1.0.0.3]; PLK2 -> FM6_ZdvihZakladacaTesnenia.PLK1 [Cable Type=PowerlinkCable, Length=10, Version=1.0.0.3]; EC1 -> M10_ManipSrobovackyOsX.EC; EC2 -> M9_ManipSrobovackyOsY.EC; EC3 -> M6_ZdvihZvaracky.EC; MT2 -> M9_ManipSrobovackyOsY.MT; MT3 -> M6_ZdvihZvaracky.MT]
  ResponseTimeout = 50
  DriveConfiguration/Module:
    McAcoposTypeID = AcoposP3TConfig
    ActivateACOPOSSimulationOnPLC = 0
  DriveConfiguration/Encoder/EncoderX41:
    InterfaceType = EnDat
  DriveConfiguration/Encoder/EncoderX42:
    InterfaceType = EnDat
  DriveConfiguration/Encoder/EncoderX43:
    InterfaceType = EnDat
  DriveConfiguration/Channel[1]:
    License = 1
  DriveConfiguration/Channel[1]/RealAxis:
    AxisReference = gAxis_3
  DriveConfiguration/Channel[1]/RealAxis/MechanicalElements/Gearbox:
    InputIsReadOnly = 0
    Input = 1
    OutputIsReadOnly = 0
    Output = 1
  DriveConfiguration/Channel[1]/RealAxis/MechanicalElements/RotaryToLinearTransformation:
    ReferenceDistanceIsReadOnly = 0
    ReferenceDistance = 10  // Rozlíšenie - 10mm/otáčku
  DriveConfiguration/Channel[1]/RealAxis/Controller:
    ModeIsReadOnly = 0
    Mode = PositionController
  DriveConfiguration/Channel[1]/RealAxis/Controller/Mode/Position:
    ProportionalGain = 473
    IntegrationTime = 0.0
    PredictionTime = 0.0004
    TotalDelayTime = 0.0004
  DriveConfiguration/Channel[1]/RealAxis/Controller/Mode/Speed:
    ProportionalGainIsReadOnly = 0
    ProportionalGain = 6.15
    IntegrationTimeIsReadOnly = 0
    IntegrationTime = 0.0
    FilterTimeIsReadOnly = 0
    FilterTime = 0.0
  DriveConfiguration/Channel[1]/RealAxis/Controller/Mode/LoopFilters:
    LoopFilter1 = NotUsed
    LoopFilter2 = NotUsed
    LoopFilter3 = NotUsed
  DriveConfiguration/Channel[1]/RealAxis/Homing:
    Mode = Direct
  DriveConfiguration/Channel[1]/RealAxis/Homing/Mode:
    Position = 0.0
    ReferencePulse = NotUsed
  DriveConfiguration/Channel[1]/RealAxis/Homing:
    RestorePositionVariable = 
  DriveConfiguration/Channel[1]/RealAxis/StopReaction:
    Quickstop = DecelerationLimit
    DriveError = DecelerationLimit
  DriveConfiguration/Channel[1]/RealAxis/MovementErrorLimits:
    PositionError = 1.0
    VelocityErrorMonitoring = Automatic1
  DriveConfiguration/Channel[1]/RealAxis:
    JerkFilter = NotUsed
  DriveConfiguration/Channel[1]/RealAxis/DigitalInputs/HomingSwitch:
    Source = NotUsed
    Level = High
  DriveConfiguration/Channel[1]/RealAxis/DigitalInputs/PositiveLimitSwitch:
    Source = NotUsed
    Level = High
  DriveConfiguration/Channel[1]/RealAxis/DigitalInputs/NegativeLimitSwitch:
    Source = NotUsed
    Level = High
  DriveConfiguration/Channel[1]/RealAxis/DigitalInputs/Trigger1:
    Source = X8Trigger1
    Level = High
  DriveConfiguration/Channel[1]/RealAxis/DigitalInputs/Trigger2:
    Source = X8Trigger2
    Level = High
  DriveConfiguration/Channel[1]/RealAxis/DigitalInputs/Quickstop:
    Input = Trigger2
  DriveConfiguration/Channel[1]/RealAxis/Simulation:
    SimulationModeOnPLC = SetValueGeneration
    SimulationModeOnACOPOS = NotUsed
  DriveConfiguration/Channel[2]:
    License = 1
  DriveConfiguration/Channel[2]/RealAxis:
    AxisReference = gAxis_4
  DriveConfiguration/Channel[2]/RealAxis/MechanicalElements/Gearbox:
    InputIsReadOnly = 0
    Input = 1
    OutputIsReadOnly = 0
    Output = 1
  DriveConfiguration/Channel[2]/RealAxis/MechanicalElements/RotaryToLinearTransformation:
    ReferenceDistanceIsReadOnly = 0
    ReferenceDistance = 10  // Rozlíšenie - 10mm/otáčku
  DriveConfiguration/Channel[2]/RealAxis/Controller:
    ModeIsReadOnly = 0
    Mode = PositionController
  DriveConfiguration/Channel[2]/RealAxis/Controller/Mode/Position:
    ProportionalGain = 556
    IntegrationTime = 0.0
    PredictionTime = 0.0004
    TotalDelayTime = 0.0004
  DriveConfiguration/Channel[2]/RealAxis/Controller/Mode/Speed:
    ProportionalGainIsReadOnly = 0
    ProportionalGain = 1.5
    IntegrationTimeIsReadOnly = 0
    IntegrationTime = 0.0
    FilterTimeIsReadOnly = 0
    FilterTime = 0.0
  DriveConfiguration/Channel[2]/RealAxis/Controller/Mode/LoopFilters:
    LoopFilter1 = NotUsed
    LoopFilter2 = NotUsed
    LoopFilter3 = NotUsed
  DriveConfiguration/Channel[2]/RealAxis/Homing:
    Mode = Direct
  DriveConfiguration/Channel[2]/RealAxis/Homing/Mode:
    Position = 0.0
    ReferencePulse = NotUsed
  DriveConfiguration/Channel[2]/RealAxis/Homing:
    RestorePositionVariable = 
  DriveConfiguration/Channel[2]/RealAxis/StopReaction:
    Quickstop = DecelerationLimit
    DriveError = DecelerationLimit
  DriveConfiguration/Channel[2]/RealAxis/MovementErrorLimits:
    PositionError = 1.0
    VelocityErrorMonitoring = Automatic1
  DriveConfiguration/Channel[2]/RealAxis:
    JerkFilter = NotUsed
  DriveConfiguration/Channel[2]/RealAxis/DigitalInputs/HomingSwitch:
    Source = NotUsed
    Level = High
  DriveConfiguration/Channel[2]/RealAxis/DigitalInputs/PositiveLimitSwitch:
    Source = NotUsed
    Level = High
  DriveConfiguration/Channel[2]/RealAxis/DigitalInputs/NegativeLimitSwitch:
    Source = NotUsed
    Level = High
  DriveConfiguration/Channel[2]/RealAxis/DigitalInputs/Trigger1:
    Source = X8Trigger1
    Level = High
  DriveConfiguration/Channel[2]/RealAxis/DigitalInputs/Trigger2:
    Source = X8Trigger2
    Level = High
  DriveConfiguration/Channel[2]/RealAxis/DigitalInputs/Quickstop:
    Input = Trigger2
  DriveConfiguration/Channel[2]/RealAxis/Simulation:
    SimulationModeOnPLC = SetValueGeneration
    SimulationModeOnACOPOS = NotUsed
  DriveConfiguration/Channel[3]:
    License = 1
  DriveConfiguration/Channel[3]/RealAxis:
    AxisReference = gAxis_5
  DriveConfiguration/Channel[3]/RealAxis/MechanicalElements/Gearbox:
    InputIsReadOnly = 0
    Input = 1
    OutputIsReadOnly = 0
    Output = 1
  DriveConfiguration/Channel[3]/RealAxis/MechanicalElements/RotaryToLinearTransformation:
    ReferenceDistanceIsReadOnly = 0
    ReferenceDistance = 10  // Rozlíšenie - 10mm/otáčku
  DriveConfiguration/Channel[3]/RealAxis/Controller:
    ModeIsReadOnly = 0
    Mode = PositionController
  DriveConfiguration/Channel[3]/RealAxis/Controller/Mode/Position:
    ProportionalGain = 405
    IntegrationTime = 0.0
    PredictionTime = 0.0004
    TotalDelayTime = 0.0004
  DriveConfiguration/Channel[3]/RealAxis/Controller/Mode/Speed:
    ProportionalGainIsReadOnly = 0
    ProportionalGain = 1.5
    IntegrationTimeIsReadOnly = 0
    IntegrationTime = 0.0
    FilterTimeIsReadOnly = 0
    FilterTime = 0.0
  DriveConfiguration/Channel[3]/RealAxis/Controller/Mode/LoopFilters:
    LoopFilter1 = NotUsed
    LoopFilter2 = NotUsed
    LoopFilter3 = NotUsed
  DriveConfiguration/Channel[3]/RealAxis/Homing:
    Mode = Direct
  DriveConfiguration/Channel[3]/RealAxis/Homing/Mode:
    Position = 0.0
    ReferencePulse = NotUsed
  DriveConfiguration/Channel[3]/RealAxis/Homing:
    RestorePositionVariable = 
  DriveConfiguration/Channel[3]/RealAxis/StopReaction:
    Quickstop = DecelerationLimit
    DriveError = DecelerationLimit
  DriveConfiguration/Channel[3]/RealAxis/MovementErrorLimits:
    PositionError = 1.0
    VelocityErrorMonitoring = Automatic1
  DriveConfiguration/Channel[3]/RealAxis:
    JerkFilter = NotUsed
  DriveConfiguration/Channel[3]/RealAxis/DigitalInputs/HomingSwitch:
    Source = NotUsed
    Level = High
  DriveConfiguration/Channel[3]/RealAxis/DigitalInputs/PositiveLimitSwitch:
    Source = NotUsed
    Level = High
  DriveConfiguration/Channel[3]/RealAxis/DigitalInputs/NegativeLimitSwitch:
    Source = NotUsed
    Level = High
  DriveConfiguration/Channel[3]/RealAxis/DigitalInputs/Trigger1:
    Source = X8Trigger1
    Level = High
  DriveConfiguration/Channel[3]/RealAxis/DigitalInputs/Trigger2:
    Source = X8Trigger2
    Level = High
  DriveConfiguration/Channel[3]/RealAxis/DigitalInputs/Quickstop:
    Input = Trigger2
  DriveConfiguration/Channel[3]/RealAxis/Simulation:
    SimulationModeOnPLC = SetValueGeneration
    SimulationModeOnACOPOS = NotUsed
FM5_ManipulatorSrobovacky : 8EI4X5MWD10.xxxx-1 v2.3.1.1  [PLK1 -> FM4_ZdvihVytahu.PLK2 [Cable Type=PowerlinkCable, Length=10, Version=1.0.0.3]; PLK2 -> VentilovyTerminal_VT4.PLK1 [Cable Type=PowerlinkCable, Length=10, Version=1.0.0.3]; EC1 -> M1.1.0.EC; EC2 -> M1.1.1.EC; MT2 -> M1.1.1.MT]
  ResponseTimeout = 50
  DriveConfiguration/Module:
    McAcoposTypeID = AcoposP3DConfig
    ActivateACOPOSSimulationOnPLC = 0
  DriveConfiguration/Encoder/EncoderX41:
    InterfaceType = EnDat
  DriveConfiguration/Encoder/EncoderX42:
    InterfaceType = EnDat
  DriveConfiguration/Channel[1]:
    License = 1
  DriveConfiguration/Channel[1]/RealAxis:
    AxisReference = gAxis_7
  DriveConfiguration/Channel[1]/RealAxis/MechanicalElements/Gearbox:
    InputIsReadOnly = 0
    Input = 1
    OutputIsReadOnly = 0
    Output = 1
  DriveConfiguration/Channel[1]/RealAxis/MechanicalElements/RotaryToLinearTransformation:
    ReferenceDistanceIsReadOnly = 0
    ReferenceDistance = 10  // Rozlíšenie - 10mm/otačku
  DriveConfiguration/Channel[1]/RealAxis/Controller:
    ModeIsReadOnly = 0
    Mode = PositionController
  DriveConfiguration/Channel[1]/RealAxis/Controller/Mode/Position:
    ProportionalGain = 534
    IntegrationTime = 0.0
    PredictionTime = 0.0004
    TotalDelayTime = 0.0004
  DriveConfiguration/Channel[1]/RealAxis/Controller/Mode/Speed:
    ProportionalGainIsReadOnly = 0
    ProportionalGain = 1.5
    IntegrationTimeIsReadOnly = 0
    IntegrationTime = 0.0
    FilterTimeIsReadOnly = 0
    FilterTime = 0.0
  DriveConfiguration/Channel[1]/RealAxis/Controller/Mode/LoopFilters:
    LoopFilter1 = NotUsed
    LoopFilter2 = NotUsed
    LoopFilter3 = NotUsed
  DriveConfiguration/Channel[1]/RealAxis/Homing:
    Mode = Direct
  DriveConfiguration/Channel[1]/RealAxis/Homing/Mode:
    Position = 0.0
    ReferencePulse = NotUsed
  DriveConfiguration/Channel[1]/RealAxis/Homing:
    RestorePositionVariable = 
  DriveConfiguration/Channel[1]/RealAxis/StopReaction:
    Quickstop = DecelerationLimit
    DriveError = DecelerationLimit
  DriveConfiguration/Channel[1]/RealAxis/MovementErrorLimits:
    PositionError = 1.0
    VelocityErrorMonitoring = Automatic1
  DriveConfiguration/Channel[1]/RealAxis:
    JerkFilter = NotUsed
  DriveConfiguration/Channel[1]/RealAxis/DigitalInputs/HomingSwitch:
    Source = NotUsed
    Level = High
  DriveConfiguration/Channel[1]/RealAxis/DigitalInputs/PositiveLimitSwitch:
    Source = NotUsed
    Level = High
  DriveConfiguration/Channel[1]/RealAxis/DigitalInputs/NegativeLimitSwitch:
    Source = NotUsed
    Level = High
  DriveConfiguration/Channel[1]/RealAxis/DigitalInputs/Trigger1:
    Source = X8Trigger1
    Level = High
  DriveConfiguration/Channel[1]/RealAxis/DigitalInputs/Trigger2:
    Source = X8Trigger2
    Level = High
  DriveConfiguration/Channel[1]/RealAxis/DigitalInputs/Quickstop:
    Input = Trigger2
  DriveConfiguration/Channel[1]/RealAxis/Simulation:
    SimulationModeOnPLC = SetValueGeneration
    SimulationModeOnACOPOS = NotUsed
  DriveConfiguration/Channel[2]:
    License = 1
  DriveConfiguration/Channel[2]/RealAxis:
    AxisReference = gAxis_8
  DriveConfiguration/Channel[2]/RealAxis/MechanicalElements/Gearbox:
    InputIsReadOnly = 0
    Input = 1
    OutputIsReadOnly = 0
    Output = 1
  DriveConfiguration/Channel[2]/RealAxis/MechanicalElements/RotaryToLinearTransformation:
    ReferenceDistanceIsReadOnly = 0
    ReferenceDistance = 10  // Rozlíšenie - 10mm/otačku
  DriveConfiguration/Channel[2]/RealAxis/Controller:
    ModeIsReadOnly = 0
    Mode = PositionController
  DriveConfiguration/Channel[2]/RealAxis/Controller/Mode/Position:
    ProportionalGain = 534
    IntegrationTime = 0.0
    PredictionTime = 0.0004
    TotalDelayTime = 0.0004
  DriveConfiguration/Channel[2]/RealAxis/Controller/Mode/Speed:
    ProportionalGainIsReadOnly = 0
    ProportionalGain = 1.5
    IntegrationTimeIsReadOnly = 0
    IntegrationTime = 0.0
    FilterTimeIsReadOnly = 0
    FilterTime = 0.0
  DriveConfiguration/Channel[2]/RealAxis/Controller/Mode/LoopFilters:
    LoopFilter1 = NotUsed
    LoopFilter2 = NotUsed
    LoopFilter3 = NotUsed
  DriveConfiguration/Channel[2]/RealAxis/Homing:
    Mode = Direct
  DriveConfiguration/Channel[2]/RealAxis/Homing/Mode:
    Position = 0.0
    ReferencePulse = NotUsed
  DriveConfiguration/Channel[2]/RealAxis/Homing:
    RestorePositionVariable = 
  DriveConfiguration/Channel[2]/RealAxis/StopReaction:
    Quickstop = DecelerationLimit
    DriveError = DecelerationLimit
  DriveConfiguration/Channel[2]/RealAxis/MovementErrorLimits:
    PositionError = 1.0
    VelocityErrorMonitoring = Automatic1
  DriveConfiguration/Channel[2]/RealAxis:
    JerkFilter = NotUsed
  DriveConfiguration/Channel[2]/RealAxis/DigitalInputs/HomingSwitch:
    Source = NotUsed
    Level = High
  DriveConfiguration/Channel[2]/RealAxis/DigitalInputs/PositiveLimitSwitch:
    Source = NotUsed
    Level = High
  DriveConfiguration/Channel[2]/RealAxis/DigitalInputs/NegativeLimitSwitch:
    Source = NotUsed
    Level = High
  DriveConfiguration/Channel[2]/RealAxis/DigitalInputs/Trigger1:
    Source = X8Trigger1
    Level = High
  DriveConfiguration/Channel[2]/RealAxis/DigitalInputs/Trigger2:
    Source = X8Trigger2
    Level = High
  DriveConfiguration/Channel[2]/RealAxis/DigitalInputs/Quickstop:
    Input = Trigger2
  DriveConfiguration/Channel[2]/RealAxis/Simulation:
    SimulationModeOnPLC = SetValueGeneration
    SimulationModeOnACOPOS = NotUsed
FM6_ZdvihZakladacaTesnenia : 8EI8X8HWS10.xxxx-1 v2.3.1.1  [PLK1 -> FM5_ManipSrobovacky_ZdvihZvarania.PLK2 [Cable Type=PowerlinkCable, Length=10, Version=1.0.0.3]; PLK2 -> FM7_PojazdZakladacaTesnenia.PLK1 [Cable Type=PowerlinkCable, Length=10, Version=1.0.0.3]; EC1 -> M4_ZdvihZakladacaTesnenia.EC]
  ResponseTimeout = 50
  DriveConfiguration/Module:
    McAcoposTypeID = AcoposP3DConfig
    ActivateACOPOSSimulationOnPLC = 0
  DriveConfiguration/Encoder/EncoderX41:
    InterfaceType = EnDat
  DriveConfiguration/Channel[1]/RealAxis:
    AxisReference = gAxis_1
  DriveConfiguration/Channel[1]/RealAxis/MechanicalElements/Gearbox:
    InputIsReadOnly = 0
    Input = 1
    OutputIsReadOnly = 0
    Output = 1
  DriveConfiguration/Channel[1]/RealAxis/MechanicalElements/RotaryToLinearTransformation:
    ReferenceDistanceIsReadOnly = 0
    ReferenceDistance = 10  // Rozlíšenie - 10mm/otačku
  DriveConfiguration/Channel[1]/RealAxis/Controller:
    ModeIsReadOnly = 0
    Mode = PositionController
  DriveConfiguration/Channel[1]/RealAxis/Controller/Mode/Position:
    ProportionalGain = 400
    IntegrationTime = 0.0
    PredictionTime = 0.0004
    TotalDelayTime = 0.0004
  DriveConfiguration/Channel[1]/RealAxis/Controller/Mode/Speed:
    ProportionalGainIsReadOnly = 0
    ProportionalGain = 2.95
    IntegrationTimeIsReadOnly = 0
    IntegrationTime = 0.0
    FilterTimeIsReadOnly = 0
    FilterTime = 0.0
  DriveConfiguration/Channel[1]/RealAxis/Controller/Mode/LoopFilters:
    LoopFilter1 = NotUsed
    LoopFilter2 = NotUsed
    LoopFilter3 = NotUsed
  DriveConfiguration/Channel[1]/RealAxis/Homing:
    Mode = Direct
  DriveConfiguration/Channel[1]/RealAxis/Homing/Mode:
    Position = 0.0
    ReferencePulse = NotUsed
  DriveConfiguration/Channel[1]/RealAxis/Homing:
    RestorePositionVariable = 
  DriveConfiguration/Channel[1]/RealAxis/StopReaction:
    Quickstop = DecelerationLimit
    DriveError = DecelerationLimit
  DriveConfiguration/Channel[1]/RealAxis/MovementErrorLimits:
    PositionError = 1.0
    VelocityErrorMonitoring = Automatic1
  DriveConfiguration/Channel[1]/RealAxis:
    JerkFilter = NotUsed
  DriveConfiguration/Channel[1]/RealAxis/DigitalInputs/HomingSwitch:
    Source = NotUsed
    Level = High
  DriveConfiguration/Channel[1]/RealAxis/DigitalInputs/PositiveLimitSwitch:
    Source = NotUsed
    Level = High
  DriveConfiguration/Channel[1]/RealAxis/DigitalInputs/NegativeLimitSwitch:
    Source = NotUsed
    Level = High
  DriveConfiguration/Channel[1]/RealAxis/DigitalInputs/Trigger1:
    Source = X8Trigger1
    Level = High
  DriveConfiguration/Channel[1]/RealAxis/DigitalInputs/Trigger2:
    Source = X8Trigger2
    Level = High
  DriveConfiguration/Channel[1]/RealAxis/DigitalInputs/Quickstop:
    Input = Trigger2
  DriveConfiguration/Channel[1]/RealAxis/Simulation:
    SimulationModeOnPLC = SetValueGeneration
    SimulationModeOnACOPOS = NotUsed
FM7_PojazdZakladacaTesnenia : 8EI4X5MWS10.xxxx-1 v2.3.1.1  [PLK1 -> FM6_ZdvihZakladacaTesnenia.PLK2 [Cable Type=PowerlinkCable, Length=10, Version=1.0.0.3]; PLK2 -> VentilovyTerminal_VT1.PLK1 [Cable Type=PowerlinkCable, Length=10, Version=1.0.0.3]; EC1 -> M5_PojazdZakladacaTesnenia.EC]
  ResponseTimeout = 50
  DriveConfiguration/Module:
    McAcoposTypeID = AcoposP3DConfig
    ActivateACOPOSSimulationOnPLC = 0
  DriveConfiguration/Encoder/EncoderX41:
    InterfaceType = EnDat
  DriveConfiguration/Channel[1]:
    License = 1
  DriveConfiguration/Channel[1]/RealAxis:
    AxisReference = gAxis_2
  DriveConfiguration/Channel[1]/RealAxis/MechanicalElements/Gearbox:
    InputIsReadOnly = 0
    Input = 10
    OutputIsReadOnly = 0
    Output = 1
  DriveConfiguration/Channel[1]/RealAxis/MechanicalElements/RotaryToLinearTransformation:
    ReferenceDistanceIsReadOnly = 0
    ReferenceDistance = 132  // Rozlíšenie - 132mm/otáčku
  DriveConfiguration/Channel[1]/RealAxis/Controller:
    ModeIsReadOnly = 0
    Mode = PositionController
  DriveConfiguration/Channel[1]/RealAxis/Controller/Mode/Position:
    ProportionalGain = 411
    IntegrationTime = 0.0
    PredictionTime = 0.0004
    TotalDelayTime = 0.0004
  DriveConfiguration/Channel[1]/RealAxis/Controller/Mode/Speed:
    ProportionalGainIsReadOnly = 0
    ProportionalGain = 0.55
    IntegrationTimeIsReadOnly = 0
    IntegrationTime = 0.0
    FilterTimeIsReadOnly = 0
    FilterTime = 0.0
  DriveConfiguration/Channel[1]/RealAxis/Controller/Mode/LoopFilters:
    LoopFilter1 = NotUsed
    LoopFilter2 = NotUsed
    LoopFilter3 = NotUsed
  DriveConfiguration/Channel[1]/RealAxis/Homing:
    Mode = Direct
  DriveConfiguration/Channel[1]/RealAxis/Homing/Mode:
    Position = 0.0
    ReferencePulse = NotUsed
  DriveConfiguration/Channel[1]/RealAxis/Homing:
    RestorePositionVariable = 
  DriveConfiguration/Channel[1]/RealAxis/StopReaction:
    Quickstop = DecelerationLimit
    DriveError = DecelerationLimit
  DriveConfiguration/Channel[1]/RealAxis/MovementErrorLimits:
    PositionError = 1.0
    VelocityErrorMonitoring = Automatic1
  DriveConfiguration/Channel[1]/RealAxis:
    JerkFilter = NotUsed
  DriveConfiguration/Channel[1]/RealAxis/DigitalInputs/HomingSwitch:
    Source = NotUsed
    Level = High
  DriveConfiguration/Channel[1]/RealAxis/DigitalInputs/PositiveLimitSwitch:
    Source = NotUsed
    Level = High
  DriveConfiguration/Channel[1]/RealAxis/DigitalInputs/NegativeLimitSwitch:
    Source = NotUsed
    Level = High
  DriveConfiguration/Channel[1]/RealAxis/DigitalInputs/Trigger1:
    Source = X8Trigger1
    Level = High
  DriveConfiguration/Channel[1]/RealAxis/DigitalInputs/Trigger2:
    Source = X8Trigger2
    Level = High
  DriveConfiguration/Channel[1]/RealAxis/DigitalInputs/Quickstop:
    Input = Trigger2
  DriveConfiguration/Channel[1]/RealAxis/Simulation:
    SimulationModeOnPLC = SetValueGeneration
    SimulationModeOnACOPOS = NotUsed
Griper4F_5F_5H_SnimacOtvoreniaZatvoreniaGripra : FBD.IOLink.GenericDeviceDTM.DTMCore.MMS xx-IOL-Mxx IODD1.1 v1.0 (OrderNumber=MMS xx-IOL-Mxx IODD1.1)  [IO-Link1 -> DS2_1.IF4]
  DtmId = f930b4fc-efc5-4e59-b1e1-e78f99b9a980
KAM_ControlUNit : FBD.Hilscher.PNIOGenDevDTM2.Control Unit V2.2 v3.14.0 (OrderNumber=Control Unit V2.2, VendorAddress=controlunit)  [PN1 -> 5ACPCI_XPNM_00.IF1]
  DtmId = 26dfd82d-0b79-4452-8dc3-6348d2a67efb
  ChannelBlocks_ecdc6902-e9b2-4869-8143-757feb0b27c0  // 2 Bytes Input <Slot 1>
  IO_InputImage_ecdc6902-e9b2-4869-8143-757feb0b27c0  // 2 Byte(s)
  ChannelBlocks_5c7b2eee-2496-439b-b6d6-de72ba0e535f  // 32 Bytes Input <Slot 2>
  IO_InputImage_5c7b2eee-2496-439b-b6d6-de72ba0e535f  // 32 Byte(s)
  ChannelBlocks_550ba9b7-d18d-4591-bef7-7b8d150ec369  // 64 Bytes Input <Slot 3>
  IO_InputImage_550ba9b7-d18d-4591-bef7-7b8d150ec369  // 64 Byte(s)
  ChannelBlocks_f5e8f8e8-0344-46d7-8c35-3852b0b4e226  // 32 Bytes Input <Slot 4>
  IO_InputImage_f5e8f8e8-0344-46d7-8c35-3852b0b4e226  // 32 Byte(s)
  ChannelBlocks_391d3c19-5eb3-4b55-b89f-b973de0fb3bf  // 64 Bytes Input <Slot 5>
  IO_InputImage_391d3c19-5eb3-4b55-b89f-b973de0fb3bf  // 64 Byte(s)
  ChannelBlocks_f852995f-546b-4cbf-bd32-76c84973c2ba  // 32 Bytes Input <Slot 6>
  IO_InputImage_f852995f-546b-4cbf-bd32-76c84973c2ba  // 32 Byte(s)
  ChannelBlocks_53e86640-3d4f-4a4b-aeb7-6a2c91a8e25d  // 64 Bytes Input <Slot 7>
  IO_InputImage_53e86640-3d4f-4a4b-aeb7-6a2c91a8e25d  // 64 Byte(s)
  ChannelBlocks_d05150e5-605c-4c7e-ac8f-d86c58b113bc  // 32 Bytes Input <Slot 8>
  IO_InputImage_d05150e5-605c-4c7e-ac8f-d86c58b113bc  // 32 Byte(s)
  ChannelBlocks_0dbe833a-b015-467a-9c23-ad398c4ac611  // 64 Bytes Input <Slot 9>
  IO_InputImage_0dbe833a-b015-467a-9c23-ad398c4ac611  // 64 Byte(s)
  ChannelBlocks_eb72156e-0593-4249-b204-fa509a5e057f  // 32 Bytes Input <Slot 10>
  IO_InputImage_eb72156e-0593-4249-b204-fa509a5e057f  // 32 Byte(s)
  ChannelBlocks_45aed417-c088-462f-bd1d-bb1c2c18bf2d  // 64 Bytes Input <Slot 11>
  IO_InputImage_45aed417-c088-462f-bd1d-bb1c2c18bf2d  // 64 Byte(s)
  ChannelBlocks_f55db729-6983-4c33-9c48-1cd40dc3f17d  // 32 Bytes Input <Slot 12>
  IO_InputImage_f55db729-6983-4c33-9c48-1cd40dc3f17d  // 32 Byte(s)
  ChannelBlocks_21169c2b-266b-40cf-b35e-180f61148f56  // 32 Bytes Input <Slot 13>
  IO_InputImage_21169c2b-266b-40cf-b35e-180f61148f56  // 32 Byte(s)
  ChannelBlocks_ad3ae690-41bc-4c51-8113-f05343acfc9b  // 32 Bytes Input <Slot 14>
  IO_InputImage_ad3ae690-41bc-4c51-8113-f05343acfc9b  // 32 Byte(s)
  ChannelBlocks_395e2464-3af9-47bf-a1c4-f46eff640543  // 64 Bytes Input <Slot 15>
  IO_InputImage_395e2464-3af9-47bf-a1c4-f46eff640543  // 64 Byte(s)
  ChannelBlocks_316771e7-db7f-4c8c-9c42-1fcc603513d9  // 32 Bytes Input <Slot 16>
  IO_InputImage_316771e7-db7f-4c8c-9c42-1fcc603513d9  // 32 Byte(s)
  ChannelBlocks_6390e492-c83e-435d-8357-46d12cfa66d2  // 64 Bytes Input <Slot 17>
  IO_InputImage_6390e492-c83e-435d-8357-46d12cfa66d2  // 64 Byte(s)
  ChannelBlocks_180ee686-5138-4850-afa8-8d5a45e14884  // 32 Bytes Input <Slot 18>
  IO_InputImage_180ee686-5138-4850-afa8-8d5a45e14884  // 32 Byte(s)
  ChannelBlocks_fd71abf0-8c89-41f4-8b97-bf62e07c27d9  // 64 Bytes Input <Slot 19>
  IO_InputImage_fd71abf0-8c89-41f4-8b97-bf62e07c27d9  // 64 Byte(s)
  ChannelBlocks_18a4a6d7-71f8-4f0c-b612-07f631054c4b  // 32 Bytes Input <Slot 20>
  IO_InputImage_18a4a6d7-71f8-4f0c-b612-07f631054c4b  // 32 Byte(s)
  ChannelBlocks_511eb5f8-a445-4331-a7a7-c895d0036a08  // 64 Bytes Input <Slot 21>
  IO_InputImage_511eb5f8-a445-4331-a7a7-c895d0036a08  // 64 Byte(s)
  ChannelBlocks_d47aa52a-7035-4ab5-b27e-782f516337c9  // 32 Bytes Input <Slot 22>
  IO_InputImage_d47aa52a-7035-4ab5-b27e-782f516337c9  // 32 Byte(s)
  ChannelBlocks_11a4f71e-9490-4fa6-a173-f76955eee4a1  // 64 Bytes Input <Slot 23>
  IO_InputImage_11a4f71e-9490-4fa6-a173-f76955eee4a1  // 64 Byte(s)
  ChannelBlocks_d23fd71c-dd4d-4f47-b681-d390591965c6  // 32 Bytes Input <Slot 24>
  IO_InputImage_d23fd71c-dd4d-4f47-b681-d390591965c6  // 32 Byte(s)
  ChannelBlocks_53804657-d470-44ec-a7a2-5696cd2137a6  // 64 Bytes Input <Slot 25>
  IO_InputImage_53804657-d470-44ec-a7a2-5696cd2137a6  // 64 Byte(s)
  ChannelBlocks_3803d2a8-8097-474e-8a2b-7f84e4f976f5  // 4 Bytes Output <Slot 26>
  IO_OutputImage_3803d2a8-8097-474e-8a2b-7f84e4f976f5  // 4 Byte(s)
  ChannelBlocks_63cae218-561f-4ebd-a86c-7fd7fe2361c0  // 4 Bytes Output <Slot 27>
  IO_OutputImage_63cae218-561f-4ebd-a86c-7fd7fe2361c0  // 4 Byte(s)
  ChannelBlocks_fe423219-bd9e-4072-884c-f33bd70f4ea3  // 4 Bytes Output <Slot 28>
  IO_OutputImage_fe423219-bd9e-4072-884c-f33bd70f4ea3  // 4 Byte(s)
  ChannelBlocks_4173e6da-c6d9-4510-bec2-190ee8648c8f  // 4 Bytes Output <Slot 29>
  IO_OutputImage_4173e6da-c6d9-4510-bec2-190ee8648c8f  // 4 Byte(s)
  ChannelBlocks_84d92d0c-a1bd-4a3b-ab94-3f3e30ea5496  // 4 Bytes Output <Slot 30>
  IO_OutputImage_84d92d0c-a1bd-4a3b-ab94-3f3e30ea5496  // 4 Byte(s)
  ChannelBlocks_41ee0638-9166-4602-835e-27eee8424401  // 4 Bytes Output <Slot 31>
  IO_OutputImage_41ee0638-9166-4602-835e-27eee8424401  // 4 Byte(s)
  ChannelBlocks_4ea2d3a4-fc47-4014-ac52-f79846c07569  // 4 Bytes Output <Slot 32>
  IO_OutputImage_4ea2d3a4-fc47-4014-ac52-f79846c07569  // 4 Byte(s)
  ChannelBlocks_ad4eb6be-d8bb-437b-804f-e773a5515d3d  // 4 Bytes Output <Slot 33>
  IO_OutputImage_ad4eb6be-d8bb-437b-804f-e773a5515d3d  // 4 Byte(s)
  ChannelBlocks_5aa70d60-5040-43b4-92aa-1669216db1d4  // 4 Bytes Output <Slot 34>
  IO_OutputImage_5aa70d60-5040-43b4-92aa-1669216db1d4  // 4 Byte(s)
  ChannelBlocks_0a00ba42-03ef-4a34-86ff-7caf6c865775  // 4 Bytes Output <Slot 35>
  IO_OutputImage_0a00ba42-03ef-4a34-86ff-7caf6c865775  // 4 Byte(s)
  ChannelBlocks_aa77839d-24e2-4c0f-ae08-c7e792622bb3  // 4 Bytes Output <Slot 36>
  IO_OutputImage_aa77839d-24e2-4c0f-ae08-c7e792622bb3  // 4 Byte(s)
  ChannelBlocks_5110b73b-bed2-4e52-95e7-3ae8a3f35cee  // 4 Bytes Output <Slot 37>
  IO_OutputImage_5110b73b-bed2-4e52-95e7-3ae8a3f35cee  // 4 Byte(s)
LeakageTester_A : FBD.Hilscher.PNIOGenDevDTM2.COMX 100XX-RE$002FPNS V3.4.19 - V3.4.x v3.4.19 (OrderNumber=COMX 100XX-RE/PNS V3.4.19 - V3.4.x, VendorAddress=ateqf6001)  [PN1 -> P3_Srobovacka_M5.PN2]
  DtmId = 93f68b6f-4f9f-4825-9dd6-ffed03a6b309
  ChannelBlocks_aff810da-93ad-4f4c-ae24-c1ba60529f89  // 64 Bytes Input <Slot 1>
  IO_InputImage_aff810da-93ad-4f4c-ae24-c1ba60529f89  // 64 Byte(s)
  ChannelBlocks_c63dfebc-1b92-4abe-a377-8275e5edb5a1  // 64 Bytes Input <Slot 2>
  IO_InputImage_c63dfebc-1b92-4abe-a377-8275e5edb5a1  // 64 Byte(s)
  ChannelBlocks_397ec51c-2b5c-451e-bc4f-b5ad16babd07  // 64 Bytes Input <Slot 3>
  IO_InputImage_397ec51c-2b5c-451e-bc4f-b5ad16babd07  // 64 Byte(s)
  ChannelBlocks_68f7ff4b-be71-4672-bab2-3928635b1302  // 64 Bytes Input <Slot 4>
  IO_InputImage_68f7ff4b-be71-4672-bab2-3928635b1302  // 64 Byte(s)
  ChannelBlocks_1dafdc3f-d861-4e38-8af1-07de8949a4a6  // 64 Bytes Output <Slot 5>
  IO_OutputImage_1dafdc3f-d861-4e38-8af1-07de8949a4a6  // 64 Byte(s)
  ChannelBlocks_8739287f-840a-44fb-aa85-4c9e176fd354  // 64 Bytes Output <Slot 6>
  IO_OutputImage_8739287f-840a-44fb-aa85-4c9e176fd354  // 64 Byte(s)
  ChannelBlocks_a4924345-ef4a-405d-89df-f807454ef77d  // 64 Bytes Output <Slot 7>
  IO_OutputImage_a4924345-ef4a-405d-89df-f807454ef77d  // 64 Byte(s)
  ChannelBlocks_fe1dc76f-2f3d-4b35-83f3-9833081ac38a  // 64 Bytes Output <Slot 8>
  IO_OutputImage_fe1dc76f-2f3d-4b35-83f3-9833081ac38a  // 64 Byte(s)
LeakageTester_B : FBD.Hilscher.PNIOGenDevDTM2.COMX 100XX-RE$002FPNS V3.4.19 - V3.4.x v3.4.19 (OrderNumber=COMX 100XX-RE/PNS V3.4.19 - V3.4.x, VendorAddress=ateqf6002)  [PN1 -> LeakageTester_A.PN2]
  DtmId = f51efb6c-bb06-4f7a-91f1-9f23b2dbe938
  ChannelBlocks_dcf2a014-9cba-4c35-bdf3-2e3e779dddd2  // 64 Bytes Input <Slot 1>
  IO_InputImage_dcf2a014-9cba-4c35-bdf3-2e3e779dddd2  // 64 Byte(s)
  ChannelBlocks_61fb6a64-30a8-4e81-8d22-591867e1cd47  // 64 Bytes Input <Slot 2>
  IO_InputImage_61fb6a64-30a8-4e81-8d22-591867e1cd47  // 64 Byte(s)
  ChannelBlocks_9f5fbe4e-efdd-46c1-b449-8d691d112cba  // 64 Bytes Input <Slot 3>
  IO_InputImage_9f5fbe4e-efdd-46c1-b449-8d691d112cba  // 64 Byte(s)
  ChannelBlocks_6b90aca8-cf2b-4c5c-bbc0-aa537b17d495  // 64 Bytes Input <Slot 4>
  IO_InputImage_6b90aca8-cf2b-4c5c-bbc0-aa537b17d495  // 64 Byte(s)
  ChannelBlocks_b2df0359-5fc7-4c8e-aeb3-77de23d401a2  // 64 Bytes Output <Slot 5>
  IO_OutputImage_b2df0359-5fc7-4c8e-aeb3-77de23d401a2  // 64 Byte(s)
  ChannelBlocks_80919c86-58a3-486d-a71b-f8644095e5f5  // 64 Bytes Output <Slot 6>
  IO_OutputImage_80919c86-58a3-486d-a71b-f8644095e5f5  // 64 Byte(s)
  ChannelBlocks_458da7c8-7676-46e3-aebc-267dfc10f1a8  // 64 Bytes Output <Slot 7>
  IO_OutputImage_458da7c8-7676-46e3-aebc-267dfc10f1a8  // 64 Byte(s)
  ChannelBlocks_58c6eb84-bfe5-4378-a7b8-f018fe1af710  // 64 Bytes Output <Slot 8>
  IO_OutputImage_58c6eb84-bfe5-4378-a7b8-f018fe1af710  // 64 Byte(s)
LeakegeTestA_SnimacPaletky_S23 : FBD.IOLink.GenericDeviceDTM.DTMCore.BIS M-404-045-401-07-S4 IODD1.0.1 v4.0 (OrderNumber=BIS M-404-045-401-07-S4 IODD1.0.1)  [IO-Link1 -> DS3_1.IF2]
  DtmId = 2c661b35-b8e3-4b8e-bb22-718cc19849cd
LeakegeTestB_SnimacPaletky_S24 : FBD.IOLink.GenericDeviceDTM.DTMCore.BIS M-404-045-401-07-S4 IODD1.0.1 v4.0 (OrderNumber=BIS M-404-045-401-07-S4 IODD1.0.1)  [IO-Link1 -> DS3_1.IF3]
  DtmId = c04d13be-5f57-42d9-9ba4-447b82f9ca3b
M1.0.0 : 8LVA23.B8015S200-0 v2.2.0.3  [EC -> FM4_ZdvihVytahu.EC1; MT -> FM4_ZdvihVytahu.MT1]
  M1/MotorParameters:
    MOTOR_AMB_TEMP_RATED = 40
M1.1.0 : 8LVA23.B9015S200-0 v2.2.0.3  [EC -> FM5_ManipulatorSrobovacky.EC1; MT -> FM5_ManipulatorSrobovacky.MT1]
  M1/MotorParameters:
    MOTOR_AMB_TEMP_RATED = 40
M1.1.1 : 8LVA23.B9015S200-0 v2.2.0.3  [EC -> FM5_ManipulatorSrobovacky.EC2; MT -> FM5_ManipulatorSrobovacky.MT2]
  M1/MotorParameters:
    MOTOR_AMB_TEMP_RATED = 40
M10_ManipSrobovackyOsX : 8LVA23.B9015S200-0 v2.2.0.3  [EC -> FM5_ManipSrobovacky_ZdvihZvarania.EC1; MT -> FM5_ManipSrobovacky_ZdvihZvarania.MT1]
  M1/MotorParameters:
    MOTOR_AMB_TEMP_RATED = 40
M26_ZdvihVytahu : 8LVA23.B8015S200-0 v2.2.0.3  [EC -> FM18_ZdvihVytahu.EC1; MT -> FM18_ZdvihVytahu.MT1]
  M1/MotorParameters:
    MOTOR_AMB_TEMP_RATED = 40
M28_ZdvihEtiketovacky : 8LVA23.B9015S200-0 v2.2.0.3  [EC -> FM19_ZdvihEtiketovacky.EC1; MT -> FM19_ZdvihEtiketovacky.MT1]
  M1/MotorParameters:
    MOTOR_AMB_TEMP_RATED = 40
M37_ManipSrobovackyOsY : 8LVA23.B9015S200-0 v2.2.0.3  [EC -> FM14_ManipSrobovacky.EC1; MT -> FM14_ManipSrobovacky.MT1]
  M1/MotorParameters:
    MOTOR_AMB_TEMP_RATED = 40
M4_ZdvihZakladacaTesnenia : 8LSA46.DB030S200-3 v2.2.0.1  [EC -> FM6_ZdvihZakladacaTesnenia.EC1; MT -> FM6_ZdvihZakladacaTesnenia.MT1]
  M1/MotorParameters:
    MOTOR_AMB_TEMP_RATED = 40
M5_PojazdZakladacaTesnenia : 8LSAA2.D9045S000-3 v2.2.0.1  [EC -> FM7_PojazdZakladacaTesnenia.EC1; MT -> FM7_PojazdZakladacaTesnenia.MT1]
  M1/MotorParameters:
    MOTOR_AMB_TEMP_RATED = 40
M6_ZdvihZvaracky : 8LVA23.B9015S200-0 v2.2.0.3  [EC -> FM5_ManipSrobovacky_ZdvihZvarania.EC3; MT -> FM5_ManipSrobovacky_ZdvihZvarania.MT3]
  M1/MotorParameters:
    MOTOR_AMB_TEMP_RATED = 40
M9_ManipSrobovackyOsY : 8LVA23.B9015S200-0 v2.2.0.3  [EC -> FM5_ManipSrobovacky_ZdvihZvarania.EC2; MT -> FM5_ManipSrobovacky_ZdvihZvarania.MT2]
  M1/MotorParameters:
    MOTOR_AMB_TEMP_RATED = 40
ModulRobot_BN1 : FBD.IOLink.GenericDeviceDTM.DTMCore.BNI IOL-309-000-K024 IODD1.0.1 v1.2 (OrderNumber=BNI IOL-309-000-K024 IODD1.0.1)  [IO-Link1 -> DS1_1.IF1]
  DtmId = c16a9b5a-9e7d-462e-acd6-1f4df0e53509
ModulRobot_BN2 : FBD.IOLink.GenericDeviceDTM.DTMCore.BNI IOL-309-000-K024 IODD1.0.1 v1.2 (OrderNumber=BNI IOL-309-000-K024 IODD1.0.1)  [IO-Link1 -> DS2_1.IF1]
  DtmId = e720d175-53bf-419b-b755-185f519cb0f3
P1_KAM3 : FBD.Hilscher.PNIOGenDevDTM2.weQube V1.4 v1.1.4 (OrderNumber=weQube V1.4, VendorAddress=cam3)  [PN1 -> KAM_ControlUNit.PN2]
  DtmId = c1dfb681-7245-4e69-b896-893c104240ba
  ChannelBlocks_80937b4a-615c-4c8d-85f5-9af72e29b7d8  // Project Number <Slot 1>
  IO_OutputImage_80937b4a-615c-4c8d-85f5-9af72e29b7d8  // 1 Byte(s)
  ChannelBlocks_011ad6fc-7215-45be-8208-bc2238c1f986  // State <Slot 2>
  IO_InputImage_011ad6fc-7215-45be-8208-bc2238c1f986  // 4 Byte(s)
  ChannelBlocks_afd5a430-5d3c-49d9-9fbf-a8960998d696  // 1 Byte Output (8 BOOL) <Slot 3>
  IO_OutputImage_afd5a430-5d3c-49d9-9fbf-a8960998d696  // 1 Byte(s)
  ChannelBlocks_f5467171-0737-4802-8377-23f82148dd12  // 64 Byte Input (2 CHAR[32]) <Slot 4>
  IO_InputImage_f5467171-0737-4802-8377-23f82148dd12  // 64 Byte(s)
  ChannelBlocks_a56ec36f-6aaf-44f7-bd86-1f8b154e6b9a  // 1 Byte Input (8 BOOL) <Slot 5>
  IO_InputImage_a56ec36f-6aaf-44f7-bd86-1f8b154e6b9a  // 1 Byte(s)
  ChannelBlocks_88039f66-4625-4e6e-b7df-6bf00e4affc6  // 16 Byte Input (4 DINT) <Slot 6>
  IO_InputImage_88039f66-4625-4e6e-b7df-6bf00e4affc6  // 16 Byte(s)
P1_KAM5 : FBD.Hilscher.PNIOGenDevDTM2.weQube V1.4 v1.1.4 (OrderNumber=weQube V1.4, VendorAddress=cam5)  [PN1 -> P1_KAM3.PN2]
  DtmId = 80fba651-141c-475b-803b-df2ebb71e074
  ChannelBlocks_da47e2b7-2559-4b41-8990-574c4f85c637  // Project Number <Slot 1>
  IO_OutputImage_da47e2b7-2559-4b41-8990-574c4f85c637  // 1 Byte(s)
  ChannelBlocks_f8c43da5-5623-45b8-97a1-792cd39e4eb9  // State <Slot 2>
  IO_InputImage_f8c43da5-5623-45b8-97a1-792cd39e4eb9  // 4 Byte(s)
  ChannelBlocks_cb67bf95-7ace-4a11-a73e-2e96bc5894ea  // 1 Byte Output (8 BOOL) <Slot 3>
  IO_OutputImage_cb67bf95-7ace-4a11-a73e-2e96bc5894ea  // 1 Byte(s)
  ChannelBlocks_c4fbc3ca-3102-4558-9131-fc390cbea9f2  // 64 Byte Input (2 CHAR[32]) <Slot 4>
  IO_InputImage_c4fbc3ca-3102-4558-9131-fc390cbea9f2  // 64 Byte(s)
  ChannelBlocks_c9323e70-2cae-44b1-857a-1409a3ff7610  // 1 Byte Input (8 BOOL) <Slot 5>
  IO_InputImage_c9323e70-2cae-44b1-857a-1409a3ff7610  // 1 Byte(s)
  ChannelBlocks_f8247db3-cef8-419d-b828-1fdaf6956654  // 16 Byte Input (4 DINT) <Slot 6>
  IO_InputImage_f8247db3-cef8-419d-b828-1fdaf6956654  // 16 Byte(s)
P2_KAM8 : FBD.Hilscher.PNIOGenDevDTM2.weQube V1.4 v1.1.4 (OrderNumber=weQube V1.4, VendorAddress=cam8)  [PN1 -> P1_KAM5.PN2]
  DtmId = d55d87c2-620b-4ac5-8e3e-6c756c2b7a96
  ChannelBlocks_f059f212-2fa3-4ee3-8beb-60b0f6785f5a  // Project Number <Slot 1>
  IO_OutputImage_f059f212-2fa3-4ee3-8beb-60b0f6785f5a  // 1 Byte(s)
  ChannelBlocks_fad9e056-eb01-4756-a331-e03aa3d0b12f  // State <Slot 2>
  IO_InputImage_fad9e056-eb01-4756-a331-e03aa3d0b12f  // 4 Byte(s)
  ChannelBlocks_af795d2f-c6a8-472a-b235-a96cc73d644b  // 1 Byte Output (8 BOOL) <Slot 3>
  IO_OutputImage_af795d2f-c6a8-472a-b235-a96cc73d644b  // 1 Byte(s)
  ChannelBlocks_05e08337-e924-4664-8784-28c230f125c3  // 64 Byte Input (2 CHAR[32]) <Slot 4>
  IO_InputImage_05e08337-e924-4664-8784-28c230f125c3  // 64 Byte(s)
  ChannelBlocks_93e7276d-4b51-48d7-a1de-8adcdf0e5d74  // 1 Byte Input (8 BOOL) <Slot 5>
  IO_InputImage_93e7276d-4b51-48d7-a1de-8adcdf0e5d74  // 1 Byte(s)
  ChannelBlocks_42b58e07-c482-48ae-8f9f-dfa47705c822  // 16 Byte Input (4 DINT) <Slot 6>
  IO_InputImage_42b58e07-c482-48ae-8f9f-dfa47705c822  // 16 Byte(s)
P2_KAM9 : FBD.Hilscher.PNIOGenDevDTM2.weQube V1.4 v1.1.4 (OrderNumber=weQube V1.4, VendorAddress=cam9)  [PN1 -> P2_KAM8.PN2]
  DtmId = 556cb3df-173f-4b65-93ae-59018d6e4b95
  ChannelBlocks_3bf3aea1-aee3-477f-bb98-b3067b13fd3b  // Project Number <Slot 1>
  IO_OutputImage_3bf3aea1-aee3-477f-bb98-b3067b13fd3b  // 1 Byte(s)
  ChannelBlocks_9fe5dc16-c3ed-461f-865b-6141d672cd55  // State <Slot 2>
  IO_InputImage_9fe5dc16-c3ed-461f-865b-6141d672cd55  // 4 Byte(s)
  ChannelBlocks_c5a0ad86-4738-4b16-ae21-e9df03187f52  // 1 Byte Output (8 BOOL) <Slot 3>
  IO_OutputImage_c5a0ad86-4738-4b16-ae21-e9df03187f52  // 1 Byte(s)
  ChannelBlocks_fef335ab-3d8a-40c8-8b22-fa9e3958cde4  // 64 Byte Input (2 CHAR[32]) <Slot 4>
  IO_InputImage_fef335ab-3d8a-40c8-8b22-fa9e3958cde4  // 64 Byte(s)
  ChannelBlocks_6479eb1b-c7e3-4ea2-aab6-832e72e9dba6  // 1 Byte Input (8 BOOL) <Slot 5>
  IO_InputImage_6479eb1b-c7e3-4ea2-aab6-832e72e9dba6  // 1 Byte(s)
  ChannelBlocks_e380a569-bd62-4c30-ab97-6436de983cf5  // 16 Byte Input (4 DINT) <Slot 6>
  IO_InputImage_e380a569-bd62-4c30-ab97-6436de983cf5  // 16 Byte(s)
P3_Srobovacka_K40 : FBD.Hilscher.PNIOGenDevDTM2.RT v0.0.0.0 (OrderNumber=RT, VendorAddress=p3-srobovacka-k40)  [PN1 -> RJ1_P2_SrobovackaMatic_M4.PN2]
  DtmId = f0183c4f-3f56-4f84-9c15-6216d67e0beb
  ChannelBlocks_8f1563f7-daef-4cdc-9755-91e87cc7356f  // Input 4 word <Slot 1>
  IO_InputImage_8f1563f7-daef-4cdc-9755-91e87cc7356f  // 8 Byte(s)
  ChannelBlocks_53490c6d-466a-4654-b596-c279f1b02e3d  // Input 4 word <Slot 2>
  IO_InputImage_53490c6d-466a-4654-b596-c279f1b02e3d  // 8 Byte(s)
  ChannelBlocks_5468e466-882a-44ec-a275-cfc8b4e035e9  // Input 4 word <Slot 3>
  IO_InputImage_5468e466-882a-44ec-a275-cfc8b4e035e9  // 8 Byte(s)
  ChannelBlocks_2f51d60d-3cec-46a7-a8d1-92c6c9f63fe4  // Input 4 word <Slot 4>
  IO_InputImage_2f51d60d-3cec-46a7-a8d1-92c6c9f63fe4  // 8 Byte(s)
  ChannelBlocks_0970dfd9-014b-46b2-bb67-b511907d5cc8  // Output 4 word <Slot 5>
  IO_OutputImage_0970dfd9-014b-46b2-bb67-b511907d5cc8  // 8 Byte(s)
  ChannelBlocks_b938d822-0f70-4f22-9641-64668ca6297f  // Output 4 word <Slot 6>
  IO_OutputImage_b938d822-0f70-4f22-9641-64668ca6297f  // 8 Byte(s)
  ChannelBlocks_8bceaa36-1e13-46a3-b487-bd1bffb761d8  // Output 4 word <Slot 7>
  IO_OutputImage_8bceaa36-1e13-46a3-b487-bd1bffb761d8  // 8 Byte(s)
  ChannelBlocks_47ba1b16-fb47-438c-9a97-702d87239931  // Output 4 word <Slot 8>
  IO_OutputImage_47ba1b16-fb47-438c-9a97-702d87239931  // 8 Byte(s)
P3_Srobovacka_M5 : FBD.Hilscher.PNIOGenDevDTM2.RT v0.0.0.0 (OrderNumber=RT, VendorAddress=p3-srobovacka-m5)  [PN1 -> P3_Srobovacka_K40.PN2]
  DtmId = 57893bde-915e-41dd-bc57-32e932aeb00c
  ChannelBlocks_390f3ebb-ea15-42a4-bf3e-8563150bdadd  // Input 4 word <Slot 1>
  IO_InputImage_390f3ebb-ea15-42a4-bf3e-8563150bdadd  // 8 Byte(s)
  ChannelBlocks_87249e8f-f6aa-47fa-ab25-d541404fdf4d  // Input 4 word <Slot 2>
  IO_InputImage_87249e8f-f6aa-47fa-ab25-d541404fdf4d  // 8 Byte(s)
  ChannelBlocks_4ec067dc-27f2-49c1-aaf2-7ac35ae462bc  // Input 4 word <Slot 3>
  IO_InputImage_4ec067dc-27f2-49c1-aaf2-7ac35ae462bc  // 8 Byte(s)
  ChannelBlocks_8caf1daa-8e7f-43ac-b229-2f64f0fd6187  // Input 4 word <Slot 4>
  IO_InputImage_8caf1daa-8e7f-43ac-b229-2f64f0fd6187  // 8 Byte(s)
  ChannelBlocks_d8fadf4f-3dbe-4493-8885-0943a1fce05c  // Output 4 word <Slot 5>
  IO_OutputImage_d8fadf4f-3dbe-4493-8885-0943a1fce05c  // 8 Byte(s)
  ChannelBlocks_f14c4b08-5b58-4c6b-b9a4-d235d4524087  // Output 4 word <Slot 6>
  IO_OutputImage_f14c4b08-5b58-4c6b-b9a4-d235d4524087  // 8 Byte(s)
  ChannelBlocks_3da9a2f3-4fe2-4e7c-9173-e1bd35dffd49  // Output 4 word <Slot 7>
  IO_OutputImage_3da9a2f3-4fe2-4e7c-9173-e1bd35dffd49  // 8 Byte(s)
  ChannelBlocks_1427dc10-635a-461e-bd6f-1200c4048a96  // Output 4 word <Slot 8>
  IO_OutputImage_1427dc10-635a-461e-bd6f-1200c4048a96  // 8 Byte(s)
P4_KAM14 : FBD.Hilscher.PNIOGenDevDTM2.weQube V1.4 v1.1.4 (OrderNumber=weQube V1.4, VendorAddress=cam14)  [PN1 -> P2_KAM9.PN2]
  DtmId = 37be806b-c4af-4935-bff4-aebcaa7f5865
  ChannelBlocks_3dd70d6c-d6d7-40b5-9610-c6be59fd2bef  // Project Number <Slot 1>
  IO_OutputImage_3dd70d6c-d6d7-40b5-9610-c6be59fd2bef  // 1 Byte(s)
  ChannelBlocks_7971ddba-fb93-4458-a135-b0b1944e5870  // State <Slot 2>
  IO_InputImage_7971ddba-fb93-4458-a135-b0b1944e5870  // 4 Byte(s)
  ChannelBlocks_197f5496-ca7c-4cb9-a206-41d6388948a5  // 1 Byte Output (8 BOOL) <Slot 3>
  IO_OutputImage_197f5496-ca7c-4cb9-a206-41d6388948a5  // 1 Byte(s)
  ChannelBlocks_2c323031-4a05-4a2a-9b3b-94983ae02249  // 64 Byte Input (2 CHAR[32]) <Slot 4>
  IO_InputImage_2c323031-4a05-4a2a-9b3b-94983ae02249  // 64 Byte(s)
  ChannelBlocks_3f0a597c-9cdf-4ca7-802e-804f69b478cf  // 1 Byte Input (8 BOOL) <Slot 5>
  IO_InputImage_3f0a597c-9cdf-4ca7-802e-804f69b478cf  // 1 Byte(s)
  ChannelBlocks_0816214e-922e-46d9-942c-e2f1b12f6f5d  // 16 Byte Input (4 DINT) <Slot 6>
  IO_InputImage_0816214e-922e-46d9-942c-e2f1b12f6f5d  // 16 Byte(s)
PC1 : 5PC910.SX02-00 v2.1.0.0
  Connector IF1:
    AssignedOperatingSystem = ARemb
  Connector IF3:
    AssignedOperatingSystem = ARemb
    ActivateDevice = 1
    Mode = Manual
    InternetAddress = 192.168.122.2
    SubnetMask = 255.255.255.0
    InaNodeNumber = 1
  Connector IF4:
    AssignedOperatingSystem = GPOS
  Connector IF10:
    OperatingSystem = ARemb
    ActivateDevice = 1
    Mode = Manual
    InternetAddress = 192.168.137.1
    SubnetMask = 255.255.255.0
  Connector IF5:
    AssignedOperatingSystem = ARemb
  Connector IF6:
    AssignedOperatingSystem = ARemb
  Connector IF7:
    AssignedOperatingSystem = ARemb
  Connector IF8:
    AssignedOperatingSystem = ARemb
  Connector IF9:
    AssignedOperatingSystem = GPOS
PS1.1 : X67PS1300 v1.0.0.0  [X2X1 -> SI1.2.X2X2 [Cable Type=X2XCable, Length=10, Version=1.0.0.3]]
PS2.1 : X67PS1300 v1.0.0.0  [X2X1 -> DM2.1_16DI/DO.X2X2 [Cable Type=X2XCable, Length=10, Version=1.0.0.3]]
PS3.1 : X67PS1300 v1.0.0.0  [X2X1 -> DI3.3_16DI.X2X2 [Cable Type=X2XCable, Length=10, Version=1.0.0.3]]
PS4.1 : X67PS1300 v1.0.0.0  [X2X1 -> DI4.1_8DI.X2X2 [Cable Type=X2XCable, Length=10, Version=1.0.0.3]]
R1_IRB120 : FBD.Hilscher.PNIOGenDevDTM2.ENERGY V1.4 v1.4 (OrderNumber=ENERGY V1.4, VendorAddress=robot-p1)  [PN1 -> AB2_1_Profinet.IF1]
  DtmId = 8eb20b82-9623-4e27-8022-3dcd0a61435e
  ChannelBlocks_be23a761-5b17-48ae-abf8-5226f03ee43f  // DI 64 bytes <Slot 1>
  IO_InputImage_be23a761-5b17-48ae-abf8-5226f03ee43f  // 64 Byte(s)
  ChannelBlocks_b1532ec0-bb1c-4408-b8fa-42838771c8b9  // DO 64 bytes <Slot 2>
  IO_OutputImage_b1532ec0-bb1c-4408-b8fa-42838771c8b9  // 64 Byte(s)
R2_IRB1200 : FBD.Hilscher.PNIOGenDevDTM2.ENERGY V1.4 v1.4 (OrderNumber=ENERGY V1.4, VendorAddress=robot-p2)  [PN1 -> R1_IRB120.PN2]
  DtmId = a2636da5-215b-46a0-aef1-ec5348bb4d2b
  ChannelBlocks_4b6f9169-7182-402e-b9d2-f260efd9d9f7  // DI 64 bytes <Slot 1>
  IO_InputImage_4b6f9169-7182-402e-b9d2-f260efd9d9f7  // 64 Byte(s)
  ChannelBlocks_bd2f4d04-4818-44a9-8413-c718b2df4356  // DO 64 bytes <Slot 2>
  IO_OutputImage_bd2f4d04-4818-44a9-8413-c718b2df4356  // 64 Byte(s)
RJ1_P2_SrobovackaMatic_M4 : FBD.Hilscher.PNIOGenDevDTM2.RT v0.0.0.0 (OrderNumber=RT, VendorAddress=p2-srobovackamatic-m4)  [PN1 -> RJ3_P2_Srobovacka_M4.PN2]
  DtmId = 8234535a-c26c-4ea4-8c11-aa00b948fab0
  ChannelBlocks_5d01e7d8-da01-4af8-90ab-19279c268217  // Input 4 word <Slot 1>
  IO_InputImage_5d01e7d8-da01-4af8-90ab-19279c268217  // 8 Byte(s)
  ChannelBlocks_6a17ae22-0d5a-4a9b-9eb5-b98bcacdc16f  // Input 4 word <Slot 2>
  IO_InputImage_6a17ae22-0d5a-4a9b-9eb5-b98bcacdc16f  // 8 Byte(s)
  ChannelBlocks_a7816c10-38f2-4dda-9321-834823b740c2  // Input 4 word <Slot 3>
  IO_InputImage_a7816c10-38f2-4dda-9321-834823b740c2  // 8 Byte(s)
  ChannelBlocks_5a5993a2-05af-45a1-9e5f-7f6f14ad3558  // Input 4 word <Slot 4>
  IO_InputImage_5a5993a2-05af-45a1-9e5f-7f6f14ad3558  // 8 Byte(s)
  ChannelBlocks_fc20f844-c8a2-49e3-834e-2127afa90704  // Output 4 word <Slot 5>
  IO_OutputImage_fc20f844-c8a2-49e3-834e-2127afa90704  // 8 Byte(s)
  ChannelBlocks_c58e44e8-f56e-4a05-bc89-cd2556593f9a  // Output 4 word <Slot 6>
  IO_OutputImage_c58e44e8-f56e-4a05-bc89-cd2556593f9a  // 8 Byte(s)
  ChannelBlocks_a48cb692-97a2-425d-b24b-4e6502c9ed7f  // Output 4 word <Slot 7>
  IO_OutputImage_a48cb692-97a2-425d-b24b-4e6502c9ed7f  // 8 Byte(s)
  ChannelBlocks_61730289-3baf-41ca-b828-007929f51b62  // Output 4 word <Slot 8>
  IO_OutputImage_61730289-3baf-41ca-b828-007929f51b62  // 8 Byte(s)
RJ2_P2_Srobovacka_M6 : FBD.Hilscher.PNIOGenDevDTM2.RT v0.0.0.0 (OrderNumber=RT, VendorAddress=p2-srobovacka-m6)  [PN1 -> RJ7_P1_Srobovacka_M4.PN2]
  DtmId = 068e73a0-6069-4b04-abde-01f818bbda4f
  ChannelBlocks_3a3b4198-c71d-43bf-998b-6716d4cf65ed  // Input 4 word <Slot 1>
  IO_InputImage_3a3b4198-c71d-43bf-998b-6716d4cf65ed  // 8 Byte(s)
  ChannelBlocks_9883f205-4a1c-4e7a-b455-26afbb897ed3  // Input 4 word <Slot 2>
  IO_InputImage_9883f205-4a1c-4e7a-b455-26afbb897ed3  // 8 Byte(s)
  ChannelBlocks_b7f2687b-9348-4f9c-a55e-d022d2d5991f  // Input 4 word <Slot 3>
  IO_InputImage_b7f2687b-9348-4f9c-a55e-d022d2d5991f  // 8 Byte(s)
  ChannelBlocks_b3284635-0bad-44d9-b1fe-64e8e0189479  // Input 4 word <Slot 4>
  IO_InputImage_b3284635-0bad-44d9-b1fe-64e8e0189479  // 8 Byte(s)
  ChannelBlocks_7050ce54-a84a-40bf-89ef-35af14d2e809  // Output 4 word <Slot 5>
  IO_OutputImage_7050ce54-a84a-40bf-89ef-35af14d2e809  // 8 Byte(s)
  ChannelBlocks_d496b44d-6163-4057-a135-fb8a36ec0817  // Output 4 word <Slot 6>
  IO_OutputImage_d496b44d-6163-4057-a135-fb8a36ec0817  // 8 Byte(s)
  ChannelBlocks_374fad07-3b64-43a5-875b-df383b88099a  // Output 4 word <Slot 7>
  IO_OutputImage_374fad07-3b64-43a5-875b-df383b88099a  // 8 Byte(s)
  ChannelBlocks_80609541-0703-4261-9393-a08bb8b3ab84  // Output 4 word <Slot 8>
  IO_OutputImage_80609541-0703-4261-9393-a08bb8b3ab84  // 8 Byte(s)
RJ3_P2_Srobovacka_M4 : FBD.Hilscher.PNIOGenDevDTM2.RT v0.0.0.0 (OrderNumber=RT, VendorAddress=p2-srobovacka-m4)  [PN1 -> RJ4_P2_Srobovacka_M5.PN2]
  DtmId = 71eb572a-e349-479b-8ca5-f9981f4f6980
  ChannelBlocks_c0c4b760-db0a-40fc-99c6-64b990e88359  // Input 4 word <Slot 1>
  IO_InputImage_c0c4b760-db0a-40fc-99c6-64b990e88359  // 8 Byte(s)
  ChannelBlocks_f4bb408f-2fa5-4f64-9369-4dd40d114b7e  // Input 4 word <Slot 2>
  IO_InputImage_f4bb408f-2fa5-4f64-9369-4dd40d114b7e  // 8 Byte(s)
  ChannelBlocks_4b709869-e9bd-4acc-82b4-3e7ce1fba065  // Input 4 word <Slot 3>
  IO_InputImage_4b709869-e9bd-4acc-82b4-3e7ce1fba065  // 8 Byte(s)
  ChannelBlocks_e19d27a5-e1cd-49cd-9af1-4c85207ef20e  // Input 4 word <Slot 4>
  IO_InputImage_e19d27a5-e1cd-49cd-9af1-4c85207ef20e  // 8 Byte(s)
  ChannelBlocks_021e5601-5e18-4674-a78e-600a48371149  // Output 4 word <Slot 5>
  IO_OutputImage_021e5601-5e18-4674-a78e-600a48371149  // 8 Byte(s)
  ChannelBlocks_1e734c6a-9936-4ede-92d0-ccaec3943c72  // Output 4 word <Slot 6>
  IO_OutputImage_1e734c6a-9936-4ede-92d0-ccaec3943c72  // 8 Byte(s)
  ChannelBlocks_0cca00b4-edc3-4b1e-a419-71976b52edba  // Output 4 word <Slot 7>
  IO_OutputImage_0cca00b4-edc3-4b1e-a419-71976b52edba  // 8 Byte(s)
  ChannelBlocks_dda1b3f1-ee81-471e-b3fa-71a6f43c8487  // Output 4 word <Slot 8>
  IO_OutputImage_dda1b3f1-ee81-471e-b3fa-71a6f43c8487  // 8 Byte(s)
RJ4_P2_Srobovacka_M5 : FBD.Hilscher.PNIOGenDevDTM2.RT v0.0.0.0 (OrderNumber=RT, VendorAddress=p2-srobovacka-m5)  [PN1 -> RJ2_P2_Srobovacka_M6.PN2]
  DtmId = 20b4d6e2-1b9b-4a23-b895-56b8382617e4
  ChannelBlocks_4dde71a8-f39c-4bfb-8cc2-8badf3cddb96  // Input 4 word <Slot 1>
  IO_InputImage_4dde71a8-f39c-4bfb-8cc2-8badf3cddb96  // 8 Byte(s)
  ChannelBlocks_b963d7ee-10cb-4e01-9138-d7569455f871  // Input 4 word <Slot 2>
  IO_InputImage_b963d7ee-10cb-4e01-9138-d7569455f871  // 8 Byte(s)
  ChannelBlocks_2ec2ba54-d2f4-4c07-b386-416ca7433072  // Input 4 word <Slot 3>
  IO_InputImage_2ec2ba54-d2f4-4c07-b386-416ca7433072  // 8 Byte(s)
  ChannelBlocks_fd2d4f12-8c20-4562-9052-bd58840ee24e  // Input 4 word <Slot 4>
  IO_InputImage_fd2d4f12-8c20-4562-9052-bd58840ee24e  // 8 Byte(s)
  ChannelBlocks_1fa7ab0c-41ab-48e9-942c-069f80e005d4  // Output 4 word <Slot 5>
  IO_OutputImage_1fa7ab0c-41ab-48e9-942c-069f80e005d4  // 8 Byte(s)
  ChannelBlocks_722ada8b-1259-4100-8d0c-f9cabf1deadd  // Output 4 word <Slot 6>
  IO_OutputImage_722ada8b-1259-4100-8d0c-f9cabf1deadd  // 8 Byte(s)
  ChannelBlocks_011b7444-62c2-42cd-9f26-fda4d5948612  // Output 4 word <Slot 7>
  IO_OutputImage_011b7444-62c2-42cd-9f26-fda4d5948612  // 8 Byte(s)
  ChannelBlocks_2716e20e-bf9f-482c-8610-b765c7d6a6a1  // Output 4 word <Slot 8>
  IO_OutputImage_2716e20e-bf9f-482c-8610-b765c7d6a6a1  // 8 Byte(s)
RJ5_P1_Srobovacka_K30 : FBD.Hilscher.PNIOGenDevDTM2.RT v0.0.0.0 (OrderNumber=RT, VendorAddress=p1-srobovacka-k30)  [PN1 -> R2_IRB1200.PN2]
  DtmId = 54f85e7e-93db-49a1-b6dd-29f0d1e2cced
  ChannelBlocks_a16bee39-a07c-46e2-9b08-1738168fe825  // Input 4 word <Slot 1>
  IO_InputImage_a16bee39-a07c-46e2-9b08-1738168fe825  // 8 Byte(s)
  ChannelBlocks_93b58e0f-75d2-4fb5-ace5-5aead8d0a898  // Input 4 word <Slot 2>
  IO_InputImage_93b58e0f-75d2-4fb5-ace5-5aead8d0a898  // 8 Byte(s)
  ChannelBlocks_fb9b3158-49c3-45d7-a35b-043216fa7ffe  // Input 4 word <Slot 3>
  IO_InputImage_fb9b3158-49c3-45d7-a35b-043216fa7ffe  // 8 Byte(s)
  ChannelBlocks_ad718db9-3945-4449-8098-cbb860637c8b  // Input 4 word <Slot 4>
  IO_InputImage_ad718db9-3945-4449-8098-cbb860637c8b  // 8 Byte(s)
  ChannelBlocks_882689f9-de29-4759-a358-f249cf8244e2  // Output 4 word <Slot 5>
  IO_OutputImage_882689f9-de29-4759-a358-f249cf8244e2  // 8 Byte(s)
  ChannelBlocks_4c935cf3-c3f3-4223-9307-729831d4dae7  // Output 4 word <Slot 6>
  IO_OutputImage_4c935cf3-c3f3-4223-9307-729831d4dae7  // 8 Byte(s)
  ChannelBlocks_7dec9e3b-3fa0-4cd2-95d6-fd01272c0df5  // Output 4 word <Slot 7>
  IO_OutputImage_7dec9e3b-3fa0-4cd2-95d6-fd01272c0df5  // 8 Byte(s)
  ChannelBlocks_e49feabf-bdf9-4869-9f0a-a21181e10023  // Output 4 word <Slot 8>
  IO_OutputImage_e49feabf-bdf9-4869-9f0a-a21181e10023  // 8 Byte(s)
RJ6_P1_Srobovacka_M5 : FBD.Hilscher.PNIOGenDevDTM2.RT v0.0.0.0 (OrderNumber=RT, VendorAddress=p1-srobovacka-m5)  [PN1 -> RJ5_P1_Srobovacka_K30.PN2]
  DtmId = 303e388f-fb7c-473d-b82b-f0cdfe95df42
  ChannelBlocks_acce06e8-3e90-4638-9e2d-5b7af71f3a87  // Input 4 word <Slot 1>
  IO_InputImage_acce06e8-3e90-4638-9e2d-5b7af71f3a87  // 8 Byte(s)
  ChannelBlocks_4f0ee3e4-db26-4ecf-a561-cc86f219bf6d  // Input 4 word <Slot 2>
  IO_InputImage_4f0ee3e4-db26-4ecf-a561-cc86f219bf6d  // 8 Byte(s)
  ChannelBlocks_5e651a88-a759-49db-bdba-709c9ecb087c  // Input 4 word <Slot 3>
  IO_InputImage_5e651a88-a759-49db-bdba-709c9ecb087c  // 8 Byte(s)
  ChannelBlocks_aa98a9d2-e5d1-4e6a-b68a-01b9d14c1e19  // Input 4 word <Slot 4>
  IO_InputImage_aa98a9d2-e5d1-4e6a-b68a-01b9d14c1e19  // 8 Byte(s)
  ChannelBlocks_97a1445d-056c-4f47-96d3-68d6890e5fec  // Output 4 word <Slot 5>
  IO_OutputImage_97a1445d-056c-4f47-96d3-68d6890e5fec  // 8 Byte(s)
  ChannelBlocks_8ec460bd-27a0-47a1-9c05-1ef827f9f2fb  // Output 4 word <Slot 6>
  IO_OutputImage_8ec460bd-27a0-47a1-9c05-1ef827f9f2fb  // 8 Byte(s)
  ChannelBlocks_e55bc582-96fe-4e55-8a8a-c6ca6b623afb  // Output 4 word <Slot 7>
  IO_OutputImage_e55bc582-96fe-4e55-8a8a-c6ca6b623afb  // 8 Byte(s)
  ChannelBlocks_6b032964-a89b-4d17-bdce-7273f731953d  // Output 4 word <Slot 8>
  IO_OutputImage_6b032964-a89b-4d17-bdce-7273f731953d  // 8 Byte(s)
RJ7_P1_Srobovacka_M4 : FBD.Hilscher.PNIOGenDevDTM2.RT v0.0.0.0 (OrderNumber=RT, VendorAddress=p1-srobovacka-m4)  [PN1 -> RJ6_P1_Srobovacka_M5.PN2]
  DtmId = d275e095-817e-4465-a46c-758d2168644c
  ChannelBlocks_a98559f4-034b-4ec8-8977-4eb834c550cc  // Input 4 word <Slot 1>
  IO_InputImage_a98559f4-034b-4ec8-8977-4eb834c550cc  // 8 Byte(s)
  ChannelBlocks_bcdd7d51-0026-4c71-b846-65df2a952e90  // Input 4 word <Slot 2>
  IO_InputImage_bcdd7d51-0026-4c71-b846-65df2a952e90  // 8 Byte(s)
  ChannelBlocks_ceb24f1a-89cf-47b4-8ba7-6569e7459ae2  // Input 4 word <Slot 3>
  IO_InputImage_ceb24f1a-89cf-47b4-8ba7-6569e7459ae2  // 8 Byte(s)
  ChannelBlocks_966a28b3-cf5f-487d-9cb4-3bd00ae77568  // Input 4 word <Slot 4>
  IO_InputImage_966a28b3-cf5f-487d-9cb4-3bd00ae77568  // 8 Byte(s)
  ChannelBlocks_d40b723f-6f36-43e8-941c-664dabbf64f6  // Output 4 word <Slot 5>
  IO_OutputImage_d40b723f-6f36-43e8-941c-664dabbf64f6  // 8 Byte(s)
  ChannelBlocks_81df151d-ae2f-4e10-89e1-731dfc559bb7  // Output 4 word <Slot 6>
  IO_OutputImage_81df151d-ae2f-4e10-89e1-731dfc559bb7  // 8 Byte(s)
  ChannelBlocks_1b087507-4962-4ec0-b86e-61a55689561d  // Output 4 word <Slot 7>
  IO_OutputImage_1b087507-4962-4ec0-b86e-61a55689561d  // 8 Byte(s)
  ChannelBlocks_e2880a6b-3981-44b9-86b7-348201ddceb8  // Output 4 word <Slot 8>
  IO_OutputImage_e2880a6b-3981-44b9-86b7-348201ddceb8  // 8 Byte(s)
SI1.1 : X67SI8103 v1.10.12.0  [X2X1 -> DI1.3_8DI.X2X2 [Cable Type=X2XCable, Length=10, Version=1.0.0.3]]
  Supervision = off
  SafeModuleID = 4
SI1.2 : X67SI8103 v1.10.12.0  [X2X1 -> DI1.1_16DI.X2X2 [Cable Type=X2XCable, Length=10, Version=1.0.0.3]]
  Supervision = off
  SafeModuleID = 5
SI2.1 : X67SI8103 v1.10.12.0  [X2X1 -> DS2_2.X2X2 [Cable Type=X2XCable, Length=10, Version=1.0.0.3]]
  Supervision = off
  SafeModuleID = 23
SI2.2 : X67SI8103 v1.10.12.0  [X2X1 -> SI2.1.X2X2 [Cable Type=X2XCable, Length=10, Version=1.0.0.3]]
  Supervision = off
  SafeModuleID = 24
SI3.1 : X67SI8103 v1.10.12.0  [X2X1 -> AB3.9_X2X.X2X1 [Cable Type=X2XCable, Length=10, Version=1.0.0.3]]
  Supervision = off
  SafeModuleID = 32
SI4.1 : X67SI8103 v1.10.12.0  [X2X1 -> PS4.1.X2X2 [Cable Type=X2XCable, Length=10, Version=1.0.0.3]]
  Supervision = off
  SafeModuleID = 43
SI4.2 : X67SI8103 v1.10.12.0  [X2X1 -> DI4.2_16DI.X2X2 [Cable Type=X2XCable, Length=10, Version=1.0.0.3]]
  Supervision = off
  SafeModuleID = 42
SL1_SafetyMaster : X20SL8100 v1.10.10.2  [PLK1 -> 0AC808.9-1.ETH2 (NodeNumber=2) [Cable Type=PowerlinkCable, Length=10, Version=1.0.0.3]; SS1 -> X20TB52.SS]
  ResponseTimeout = 50
  Supervision = off
  SafeProject = SafeLOGIC-1
  SafeDesigner = 4.3.4.4
  UnsafeOutputBOOLs = 64
  UnsafeInputBOOLs = 64
SkrutkovacMatic_VysunutieHrotuSkrutkovacky_IOS7 : FBD.IOLink.GenericDeviceDTM.DTMCore.Magnetic Cylinder Sensors IODD1.1 v1.3 (OrderNumber=Magnetic Cylinder Sensors IODD1.1)  [IO-Link1 -> DS2_1.IF3]
  DtmId = 715e7600-8bd3-4dba-a433-f8a9f1959dfc
SkrutkovackaK30_VysunutieHrotu_IOS8 : FBD.IOLink.GenericDeviceDTM.DTMCore.Magnetic Cylinder Sensors IODD1.1 v1.3 (OrderNumber=Magnetic Cylinder Sensors IODD1.1)  [IO-Link1 -> DS1_2.IF1]
  DtmId = 4779cc4d-2790-4fae-a1a3-f7e2ee2d3f8d
SkrutkovackaK40_VysunutieHrotuSkrutkovacky_IOS11 : FBD.IOLink.GenericDeviceDTM.DTMCore.Magnetic Cylinder Sensors IODD1.1 v1.3 (OrderNumber=Magnetic Cylinder Sensors IODD1.1)  [IO-Link1 -> DS3_3.IF1]
  DtmId = 996746c4-4602-4290-a6aa-ffe1793630dd
SkrutkovackaM4_VysunutieHrotuSkrutkovacky_IOS4 : FBD.IOLink.GenericDeviceDTM.DTMCore.Magnetic Cylinder Sensors IODD1.1 v1.3 (OrderNumber=Magnetic Cylinder Sensors IODD1.1)  [IO-Link1 -> DS2_3.IF2]
  DtmId = b7288bc3-72ce-4be0-a9b0-0d559dd3a3e1
SkrutkovackaM4_VysunutieHrotu_IOS9 : FBD.IOLink.GenericDeviceDTM.DTMCore.Magnetic Cylinder Sensors IODD1.1 v1.3 (OrderNumber=Magnetic Cylinder Sensors IODD1.1)  [IO-Link1 -> DS1_2.IF2]
  DtmId = 3a1249a2-26c4-4f4a-97b9-2452d1be8397
SkrutkovackaM5_VysunutieHrotuSkrutkovacky_IOS12 : FBD.IOLink.GenericDeviceDTM.DTMCore.Magnetic Cylinder Sensors IODD1.1 v1.3 (OrderNumber=Magnetic Cylinder Sensors IODD1.1)  [IO-Link1 -> DS3_3.IF2]
  DtmId = 3e16b5bc-f884-4c83-910a-31c26e95057b
SkrutkovackaM5_VysunutieHrotuSkrutkovacky_IOS5 : FBD.IOLink.GenericDeviceDTM.DTMCore.Magnetic Cylinder Sensors IODD1.1 v1.3 (OrderNumber=Magnetic Cylinder Sensors IODD1.1)  [IO-Link1 -> DS2_3.IF3]
  DtmId = ea9fb762-e59c-4a66-8c75-1a95d0c31415
SkrutkovackaM5_VysunutieHrotu_IOS10 : FBD.IOLink.GenericDeviceDTM.DTMCore.Magnetic Cylinder Sensors IODD1.1 v1.3 (OrderNumber=Magnetic Cylinder Sensors IODD1.1)  [IO-Link1 -> DS1_2.IF3]
  DtmId = 0d8b74b1-204b-4f4b-bddd-910e6e24c19e
SkrutkovackaM6_VysunutieHrotuSkrutkovacky_IOS3 : FBD.IOLink.GenericDeviceDTM.DTMCore.Magnetic Cylinder Sensors IODD1.1 v1.3 (OrderNumber=Magnetic Cylinder Sensors IODD1.1)  [IO-Link1 -> DS2_3.IF1]
  DtmId = 5ec77f1b-7475-4bfa-9e17-f45b7cc319ec
SnimacTlakuLeakeTestA_S26 : FBD.IOLink.GenericDeviceDTM.DTMCore.BSP00PU IODD1.1 v1.1 (OrderNumber=BSP00PU IODD1.1)  [IO-Link1 -> DS3_2.IF1]
  DtmId = 31e4389b-1594-481b-992c-dc0f2df3747c
SnimacTlakuLeakeTestB_S27 : FBD.IOLink.GenericDeviceDTM.DTMCore.BSP00PU IODD1.1 v1.1 (OrderNumber=BSP00PU IODD1.1)  [IO-Link1 -> DS3_2.IF2]
  DtmId = bf3fc145-622c-459b-8e01-a91c90950947
StoperEtiketovacky_SnimacPaletky_S12 : FBD.IOLink.GenericDeviceDTM.DTMCore.BIS M-404-045-401-07-S4 IODD1.0.1 v4.0 (OrderNumber=BIS M-404-045-401-07-S4 IODD1.0.1)  [IO-Link1 -> DS4_1.IF3]
  DtmId = 879da402-b547-4dcc-8a67-c8676b554ee1
StoperFunkcnyTestA_SnimacPaletky_S10 : FBD.IOLink.GenericDeviceDTM.DTMCore.BIS M-404-045-401-07-S4 IODD1.0.1 v4.0 (OrderNumber=BIS M-404-045-401-07-S4 IODD1.0.1)  [IO-Link1 -> DS4_1.IF1]
  DtmId = 335848d8-1b8e-405c-a7c7-3b121369d6ec
StoperFunkcnyTestB_SnimacPaletky_S11 : FBD.IOLink.GenericDeviceDTM.DTMCore.BIS M-404-045-401-07-S4 IODD1.0.1 v4.0 (OrderNumber=BIS M-404-045-401-07-S4 IODD1.0.1)  [IO-Link1 -> DS4_1.IF2]
  DtmId = 8f53176d-fc28-468c-95cf-d799fa2a3e2f
StoperSkrutkovaniaMatic_SnimacPaletky_S7 : FBD.IOLink.GenericDeviceDTM.DTMCore.BIS M-404-045-401-07-S4 IODD1.0.1 v4.0 (OrderNumber=BIS M-404-045-401-07-S4 IODD1.0.1)  [IO-Link1 -> DS2_2.IF2]
  DtmId = 748b1a3b-534b-497e-b703-cffcc7a9ab85
StoperSkrutkovania_SnimacPaletky_S22 : FBD.IOLink.GenericDeviceDTM.DTMCore.BIS M-404-045-401-07-S4 IODD1.0.1 v4.0 (OrderNumber=BIS M-404-045-401-07-S4 IODD1.0.1)  [IO-Link1 -> DS3_1.IF1]
  DtmId = a02b6854-9dbe-4f88-be3e-1320b4aeffec
StoperSrobovania_SnimacPaletky_S16 : FBD.IOLink.GenericDeviceDTM.DTMCore.BIS M-404-045-401-07-S4 IODD1.0.1 v4.0 (OrderNumber=BIS M-404-045-401-07-S4 IODD1.0.1)  [IO-Link1 -> DS1_1.IF4]
  DtmId = 14f46eb3-09cd-449e-a308-b3cd2b497734
StoperSrobovania_SnimacPaletky_S8 : FBD.IOLink.GenericDeviceDTM.DTMCore.BIS M-404-045-401-07-S4 IODD1.0.1 v4.0 (OrderNumber=BIS M-404-045-401-07-S4 IODD1.0.1)  [IO-Link1 -> DS2_2.IF3]
  DtmId = e08233f0-b813-44d1-90f7-8d1dd5337b2a
StoperZakladaniaTesnenia_SnimacPaletky_S6 : FBD.IOLink.GenericDeviceDTM.DTMCore.BIS M-404-045-401-07-S4 IODD1.0.1 v4.0 (OrderNumber=BIS M-404-045-401-07-S4 IODD1.0.1)  [IO-Link1 -> DS2_2.IF1]
  DtmId = 1fe25137-3686-4f60-8fd0-fa0540cf0608
StoperZvarania_SnimacPaletky_S9 : FBD.IOLink.GenericDeviceDTM.DTMCore.BIS M-404-045-401-07-S4 IODD1.0.1 v4.0 (OrderNumber=BIS M-404-045-401-07-S4 IODD1.0.1)  [IO-Link1 -> DS2_2.IF4]
  DtmId = 37bbaa9a-fc5e-4930-9e1d-a96b25094715
VentilovyTerminal_VT1 : FBE.FFFF0007_EX260-SPL1 v1.0 (OrderNumber=EX260-SPL1)  [PLK1 -> FM7_PojazdZakladacaTesnenia.PLK2 [Cable Type=PowerlinkCable, Length=10, Version=1.0.0.3]; PLK2 -> VentilovyTerminal_VT2.PLK1 [Cable Type=PowerlinkCable, Length=10, Version=1.0.0.3]]
  Supervision = off
  ResponseTimeout = 50
VentilovyTerminal_VT2 : FBE.FFFF0007_EX260-SPL1 v1.0 (OrderNumber=EX260-SPL1)  [PLK1 -> VentilovyTerminal_VT1.PLK2 [Cable Type=PowerlinkCable, Length=10, Version=1.0.0.3]; PLK2 -> VentilovyTerminal_VT3.PLK1 [Cable Type=PowerlinkCable, Length=10, Version=1.0.0.3]]
  Supervision = off
  ResponseTimeout = 50
VentilovyTerminal_VT3 : FBE.FFFF0007_EX260-SPL1 v1.0 (OrderNumber=EX260-SPL1)  [PLK1 -> VentilovyTerminal_VT2.PLK2 [Cable Type=PowerlinkCable, Length=10, Version=1.0.0.3]]
  Supervision = off
  ResponseTimeout = 50
VentilovyTerminal_VT4 : FBE.FFFF0007_EX260-SPL1 v1.0 (OrderNumber=EX260-SPL1)  [PLK1 -> FM5_ManipulatorSrobovacky.PLK2 [Cable Type=PowerlinkCable, Length=10, Version=1.0.0.3]; PLK2 -> VentilovyTerminal_VT5.PLK1 [Cable Type=PowerlinkCable, Length=10, Version=1.0.0.3]]
  Supervision = off
  ResponseTimeout = 50
VentilovyTerminal_VT5 : FBE.FFFF0007_EX260-SPL1 v1.0 (OrderNumber=EX260-SPL1)  [PLK1 -> VentilovyTerminal_VT4.PLK2 [Cable Type=PowerlinkCable, Length=10, Version=1.0.0.3]]
  Supervision = off
  ResponseTimeout = 50
VentilovyTerminal_VT6 : FBE.FFFF0007_EX260-SPL1 v1.0 (OrderNumber=EX260-SPL1)  [PLK1 -> FM14_ManipSrobovacky.PLK2 [Cable Type=PowerlinkCable, Length=10, Version=1.0.0.3]; PLK2 -> VentilovyTerminal_VT7.PLK1 [Cable Type=PowerlinkCable, Length=10, Version=1.0.0.3]]
  Supervision = off
  ResponseTimeout = 50
VentilovyTerminal_VT7 : FBE.FFFF0007_EX260-SPL1 v1.0 (OrderNumber=EX260-SPL1)  [PLK1 -> VentilovyTerminal_VT6.PLK2 [Cable Type=PowerlinkCable, Length=10, Version=1.0.0.3]]
  Supervision = off
  ResponseTimeout = 50
VentilovyTerminal_VT8 : FBE.FFFF0007_EX260-SPL1 v1.0 (OrderNumber=EX260-SPL1)  [PLK1 -> FM18_ZdvihVytahu.PLK2 [Cable Type=PowerlinkCable, Length=10, Version=1.0.0.3]]
  Supervision = off
  ResponseTimeout = 50
Vytah_BannerPotvrdeniaObsluhy_SB10 : FBD.IOLink.GenericDeviceDTM.DTMCore.K50 Pro Device IODD1.1 v1.3 (OrderNumber=K50 Pro Device IODD1.1)  [IO-Link1 -> DS4_2.IF1]
  DtmId = 634f8f05-67f7-4553-99b2-588c89e53489
Vytah_BannerPotvrdeniaObsluhy_SB11 : FBD.IOLink.GenericDeviceDTM.DTMCore.K50 Pro Device IODD1.1 v1.3 (OrderNumber=K50 Pro Device IODD1.1)  [IO-Link1 -> DS1_1.IF2]
  DtmId = 501ead61-16d6-479a-8c72-f9baa0e8a6bf
Vytah_SnimacPaletky_S13 : FBD.IOLink.GenericDeviceDTM.DTMCore.BIS M-404-045-401-07-S4 IODD1.0.1 v4.0 (OrderNumber=BIS M-404-045-401-07-S4 IODD1.0.1)  [IO-Link1 -> DS4_2.IF2]
  DtmId = c1e54278-c882-402c-94ee-fb6ed3aa02f1
Vytah_SnimacPaletky_S19 : FBD.IOLink.GenericDeviceDTM.DTMCore.BIS M-404-045-401-07-S4 IODD1.0.1 v4.0 (OrderNumber=BIS M-404-045-401-07-S4 IODD1.0.1)  [IO-Link1 -> DS1_1.IF3]
  DtmId = f9cd6e35-af4a-42f2-af08-71c2d09ca6cd
X20BB81 : X20BB81 v1.1.0.0
X20BB81a : X20BB81 v1.1.0.0
X20BB81b : X20BB81 v1.1.0.0
X20BB81c : X20BB81 v1.1.0.0
X20BM11 : X20BM11 v1.1.0.0  [X2X1 -> X20BM33d.X2X2]
X20BM11a : X20BM11 v1.1.0.0  [X2X1 -> X20BM11.X2X2]
X20BM11b : X20BM11 v1.1.0.0  [X2X1 -> X20BM11a.X2X2]
X20BM11c : X20BM11 v1.1.0.0  [X2X1 -> X20BM11b.X2X2]
X20BM11d : X20BM11 v1.1.0.0  [X2X1 -> X20BM33h.X2X2]
X20BM11e : X20BM11 v1.1.0.0  [X2X1 -> X20BM11d.X2X2]
X20BM11f : X20BM11 v1.1.0.0  [X2X1 -> X20BB81b.IF1]
X20BM11g : X20BM11 v1.1.0.0  [X2X1 -> X20BM11f.X2X2]
X20BM11h : X20BM11 v1.1.0.0  [X2X1 -> X20BM11c.X2X2]
X20BM11i : X20BM11 v1.1.0.0  [X2X1 -> X20BM11m.X2X2]
X20BM11j : X20BM11 v1.1.0.0  [X2X1 -> X20BM33f.X2X2]
X20BM11k : X20BM11 v1.1.0.0  [X2X1 -> X20BM11o.X2X2]
X20BM11l : X20BM11 v1.1.0.0  [X2X1 -> X20BM11e.X2X2]
X20BM11m : X20BM11 v1.1.0.0  [X2X1 -> X20BM11l.X2X2]
X20BM11n : X20BM11 v1.1.0.0  [X2X1 -> X20BM33g.X2X2]
X20BM11o : X20BM11 v1.1.0.0  [X2X1 -> X20BM11n.X2X2]
X20BM33 : X20BM33 v1.1.0.0  [X2X1 -> X20BB81.IF1]
X20BM33a : X20BM33 v1.1.0.0  [X2X1 -> X20BB81a.IF1]
X20BM33b : X20BM33 v1.1.0.0  [X2X1 -> X20BM11g.X2X2]
X20BM33c : X20BM33 v1.1.0.0  [X2X1 -> X20BB81c.IF1]
X20BM33d : X20BM33 v1.1.0.0  [X2X1 -> X20BM33.X2X2]
X20BM33e : X20BM33 v1.1.0.0  [X2X1 -> X20BM33a.X2X2]
X20BM33f : X20BM33 v1.1.0.0  [X2X1 -> X20BM33b.X2X2]
X20BM33g : X20BM33 v1.1.0.0  [X2X1 -> X20BM33c.X2X2]
X20BM33h : X20BM33 v1.1.0.0  [X2X1 -> X20BM33e.X2X2]
X20MK0211 : X20MK0211 v1.0.0.3  [SL -> SL1_SafetyMaster.SL1]
X20TB12 : X20TB12 v1.0.0.0
X20TB12a : X20TB12 v1.0.0.0
X20TB12b : X20TB12 v1.0.0.0
X20TB12c : X20TB12 v1.0.0.0
X20TB12d : X20TB12 v1.0.0.0
X20TB12e : X20TB12 v1.0.0.0
X20TB12f : X20TB12 v1.0.0.0
X20TB12g : X20TB12 v1.0.0.0
X20TB1F : X20TB1F v1.0.0.0
X20TB1F1 : X20TB1F v1.0.0.0
X20TB1F10 : X20TB1F v1.0.0.0
X20TB1F11 : X20TB1F v1.0.0.0
X20TB1F2 : X20TB1F v1.0.0.0
X20TB1F3 : X20TB1F v1.0.0.0
X20TB1F4 : X20TB1F v1.0.0.0
X20TB1F5 : X20TB1F v1.0.0.0
X20TB1F6 : X20TB1F v1.0.0.0
X20TB1F7 : X20TB1F v1.0.0.0
X20TB1F8 : X20TB1F v1.0.0.0
X20TB1F9 : X20TB1F v1.0.0.0
X20TB52 : X20TB52 v1.0.0.2
X20TB52a : X20TB52 v1.0.0.2
X20TB52b : X20TB52 v1.0.0.2
X20TB52c : X20TB52 v1.0.0.2
X20TB52d : X20TB52 v1.0.0.2
X20TB52e : X20TB52 v1.0.0.2
X20TB52f : X20TB52 v1.0.0.2
X20TB52g : X20TB52 v1.0.0.2
X20TB52h : X20TB52 v1.0.0.2
X20TB52i : X20TB52 v1.0.0.2
X20TB52j : X20TB52 v1.0.0.2
X20TB52k : X20TB52 v1.0.0.2
X20TB52l : X20TB52 v1.0.0.2
X20TB52m : X20TB52 v1.0.0.2
ZakladacTesnenia_BannerPotvrdeniaObsluhy_SB7 : FBD.IOLink.GenericDeviceDTM.DTMCore.K50 Pro Device IODD1.1 v1.3 (OrderNumber=K50 Pro Device IODD1.1)  [IO-Link1 -> DS2_1.IF2]
  DtmId = dbb14531-e218-45c6-abe8-6a40ae98327a
```
